// TwinCAT 3 PLC project TcUnit
// Title: TcUnit
// Company: www.tcunit.org
// Author: Jakob Sagatowski and contributors
// ProjectVersion: 1.3.2
// Description: TwinCAT unit testing framework. Documentation and examples are available at www.tcunit.org
// ProgramVersion: 3.1.4022.2
// libraries:
//   SysDir, * (System)
//   SysFile, * (System)
//   Tc2_Standard, * (Beckhoff Automation GmbH)
//   Tc2_System, * (Beckhoff Automation GmbH)
//   Tc2_Utilities, * (Beckhoff Automation GmbH)
//   Base Interfaces,newest,System
// project tree:
//   DUTs/ E_AssertionType.TcDUT, E_XmlError.TcDUT, ST_AdsLogStringMessage.TcDUT, ST_AssertResult.TcDUT, ST_AssertResultInstances.TcDUT, ST_AssertArrayResult.TcDUT, ST_AssertArrayResultInstances.TcDUT, ST_TestCaseResult.TcDUT, ST_TestSuiteResult.TcDUT, ST_TestSuiteResults.TcDUT, U_ExpectedOrActual.TcDUT
//   GVLs/ GVL_Param_TcUnit.TcGVL, GVL_TcUnit.TcGVL
//   ITFs/ I_AssertMessageFormatter.TcIO, I_TestResultLogger.TcIO, I_TestResults.TcIO
//   POUs/ FB_AdsAssertMessageFormatter.TcPOU, FB_AdsLogStringMessageFifoQueue.TcPOU, FB_AdsTestResultLogger.TcPOU, FB_FileControl.TcPOU, FB_StreamBuffer.TcPOU, FB_xUnitXmlPublisher.TcPOU, FB_TestResults.TcPOU, FB_AdjustAssertFailureMessageToMaxAllowedLength.TcPOU, FB_AssertResultStatic.TcPOU, FB_AssertArrayResultStatic.TcPOU, FB_TcUnitRunner.TcPOU, FB_Test.TcPOU, FB_TestSuite.TcPOU, FB_XmlControl.TcPOU
//   POUs/Functions/ F_AnyToUnionValue.TcPOU, F_AnyTypeClassToString.TcPOU, F_AssertionTypeToString.TcPOU, F_GetCpuCounterAs64bit.TcPOU, F_GetTestSuiteNameFromTestInstancePath.TcPOU, F_IsAnyEqualToUnionValue.TcPOU, F_RemoveInstancePathAndProjectNameFromTestInstancePath.TcPOU, IS_TEST_FINISHED.TcPOU, RUN.TcPOU, RUN_IN_SEQUENCE.TcPOU, TCUNIT_ADSLOGSTR.TcPOU, TEST.TcPOU, TEST_FINISHED.TcPOU, TEST_FINISHED_NAMED.TcPOU, TEST_ORDERED.TcPOU
//   POUs/Functions/WRITE_PROTECTED_/ WRITE_PROTECTED_BOOL.TcPOU, WRITE_PROTECTED_BYTE.TcPOU, WRITE_PROTECTED_DATE.TcPOU, WRITE_PROTECTED_DATE_AND_TIME.TcPOU, WRITE_PROTECTED_DINT.TcPOU, WRITE_PROTECTED_DWORD.TcPOU, WRITE_PROTECTED_INT.TcPOU, WRITE_PROTECTED_LREAL.TcPOU, WRITE_PROTECTED_REAL.TcPOU, WRITE_PROTECTED_SINT.TcPOU, WRITE_PROTECTED_STRING.TcPOU, WRITE_PROTECTED_WSTRING.TcPOU, WRITE_PROTECTED_TIME.TcPOU, WRITE_PROTECTED_TIME_OF_DAY.TcPOU, WRITE_PROTECTED_UDINT.TcPOU, WRITE_PROTECTED_UINT.TcPOU, WRITE_PROTECTED_ULINT.TcPOU, WRITE_PROTECTED_LWORD.TcPOU, WRITE_PROTECTED_LINT.TcPOU, WRITE_PROTECTED_USINT.TcPOU, WRITE_PROTECTED_WORD.TcPOU
//   Version/ Global_Version.TcGVL

// ---- DUTs/E_AssertionType.TcDUT
{attribute 'qualified_only'}
{attribute 'strict'}
TYPE E_AssertionType :
(
    Type_UNDEFINED := 0,
    Type_ANY,

    // Primitive types
    Type_BOOL,
    Type_BYTE,
    Type_DATE,
    Type_DATE_AND_TIME,
    Type_DINT,
    Type_DWORD,
    Type_INT,
    Type_LINT,
    Type_LREAL,
    Type_LTIME,
    Type_LWORD,
    Type_REAL,
    Type_SINT,
    Type_STRING,
    Type_TIME,
    Type_TIME_OF_DAY,
    Type_UDINT,
    Type_UINT,
    Type_ULINT,
    Type_USINT,
    Type_WORD,
    Type_WSTRING,

    // Array types
    Type_Array2D_LREAL,
    Type_Array2D_REAL,
    Type_Array3D_LREAL,
    Type_Array3D_REAL,
    Type_Array_BOOL,
    Type_Array_BYTE,
    Type_Array_DINT,
    Type_Array_DWORD,
    Type_Array_INT,
    Type_Array_LINT,
    Type_Array_LREAL,
    Type_Array_LWORD,
    Type_Array_REAL,
    Type_Array_SINT,
    Type_Array_UDINT,
    Type_Array_UINT,
    Type_Array_ULINT,
    Type_Array_USINT,
    Type_Array_WORD
) BYTE;
END_TYPE

// ---- DUTs/E_XmlError.TcDUT
{attribute 'qualified_only'}
{attribute 'strict'}
TYPE E_XmlError :
(
    Ok := 0,
    ErrorMaxBufferLen := 1,
    ErrorStringLen := 2,
    Error := 3
) BYTE;
END_TYPE

// ---- DUTs/ST_AdsLogStringMessage.TcDUT
{attribute 'pack_mode' := '1'}
TYPE ST_AdsLogStringMessage :
STRUCT
	MsgCtrlMask : DWORD;
    MsgFmtStr : T_MaxString;
    StrArg : T_MaxString;
END_STRUCT
END_TYPE

// ---- DUTs/ST_AssertResult.TcDUT
TYPE ST_AssertResult :
STRUCT
    Expected : U_ExpectedOrActual;
    Actual : U_ExpectedOrActual;
    Message : T_MaxString;
    TestInstancePath : T_MaxString;
END_STRUCT
END_TYPE

// ---- DUTs/ST_AssertResultInstances.TcDUT
TYPE ST_AssertResultInstances :
STRUCT
    AssertResult : ST_AssertResult;
    DetectionCount : UINT; // Number of instances of the "AssertResult"
    DetectionCountThisCycle : UINT; // Number of instance of the "AssertResult" in this specific PLC-cycle
END_STRUCT
END_TYPE

// ---- DUTs/ST_AssertArrayResult.TcDUT
TYPE ST_AssertArrayResult :
STRUCT
    ExpectedsSize : UDINT; // Size in bytes of the expecteds-array
    ExpectedsTypeClass : IBaseLibrary.TypeClass; // The data type of the expecteds-array
    ActualsSize : UDINT; // Size in bytes of the actuals-array
    ActualsTypeClass : IBaseLibrary.TypeClass; // The data type of the actuals-array
    Message : T_MaxString;
    TestInstancePath : T_MaxString;
END_STRUCT
END_TYPE

// ---- DUTs/ST_AssertArrayResultInstances.TcDUT
TYPE ST_AssertArrayResultInstances :
STRUCT
    AssertArrayResult : ST_AssertArrayResult;
    DetectionCount : UINT; // Number of instances of the "AssertArrayResult"
    DetectionCountThisCycle : UINT; // Number of instance of the "AssertArrayResult" in this specific PLC-cycle
END_STRUCT
END_TYPE

// ---- DUTs/ST_TestCaseResult.TcDUT
TYPE ST_TestCaseResult :
STRUCT
    TestName : T_MaxString;
    TestClassName : T_MaxString;
    TestIsFailed : BOOL;
    TestIsSkipped : BOOL;
    FailureMessage : T_MaxString;
    FailureAssertion : Tc2_System.T_MaxString;
    FailureType : E_AssertionType;
    NumberOfAsserts : UINT;
    Duration : LREAL; // in seconds
END_STRUCT
END_TYPE

// ---- DUTs/ST_TestSuiteResult.TcDUT
TYPE ST_TestSuiteResult :
STRUCT
    Name : T_MaxString; // Full class name
    Identity : UINT(0..GVL_Param_TcUnit.MaxNumberOfTestSuites); // Should be 0..GVL_Param_TcUnit.MaxNumberOfTestSuites-1 but gives unknown compiler error
    NumberOfTests : UINT(0..GVL_Param_TcUnit.MaxNumberOfTestsForEachTestSuite);
    NumberOfFailedTests : UINT(0..GVL_Param_TcUnit.MaxNumberOfTestsForEachTestSuite);
    Duration : LREAL; // In seconds
    TestCaseResults : ARRAY[1..GVL_Param_TcUnit.MaxNumberOfTestsForEachTestSuite] OF ST_TestCaseResult;
END_STRUCT
END_TYPE

// ---- DUTs/ST_TestSuiteResults.TcDUT
TYPE ST_TestSuiteResults :
STRUCT
    // General test results
    NumberOfTestSuites : UINT; // The total number of test suites
    NumberOfTestCases : UINT; // The total number of test cases (for all test suites)
    NumberOfSuccessfulTestCases : UINT; // The total number of test cases that had all ASSERTS successful
    NumberOfFailedTestCases : UINT; // The total number of test cases that had at least one ASSERT failed
    Duration : LREAL; // Duration it took for all test suites to finish, in seconds

    // Test results for each individiual test suite
    TestSuiteResults : ARRAY[1..GVL_Param_TcUnit.MaxNumberOfTestSuites] OF ST_TestSuiteResult;
END_STRUCT
END_TYPE

// ---- DUTs/U_ExpectedOrActual.TcDUT
TYPE U_ExpectedOrActual :
UNION
    boolExpectedOrActual : BOOL;
    bitExpectedOrActual : BIT;
    byteExpectedOrActual : BYTE;
    dwordExpectedOrActual : DWORD;
    lwordExpectedOrActual : LWORD;
    stringExpectedOrActual : T_MaxString;
    udintExpectedOrActual : UDINT;
    uintExpectedOrActual : UINT;
    usintExpectedOrActual : USINT;
    sintExpectedOrActual : SINT;
    intExpectedOrActual : INT;
    wordExpectedOrActual : WORD;
    dintExpectedOrActual : DINT;
    lintExpectedOrActual : LINT;
    ulintExpectedOrActual : ULINT;
    realExpectedOrActual : REAL;
    lrealExpectedOrActual : LREAL;
    wstringExpectedOrActual : WSTRING(255);
    timeExpectedOrActual : TIME;
    ltimeExpectedOrActual : LTIME;
    dateExpectedOrActual : DATE;
    dateandtimeExpectedOrActual : DATE_AND_TIME;
    timeofdayExpectedOrActual : TIME_OF_DAY;
END_UNION
END_TYPE

// ---- GVLs/GVL_Param_TcUnit.TcGVL
{attribute 'qualified_only'}
VAR_GLOBAL CONSTANT
    MaxNumberOfTestSuites : UINT := 1000;
    MaxNumberOfTestsForEachTestSuite : UINT := 100;
    MaxNumberOfAssertsForEachTestSuite : UINT := 1000;

    (* TcUnit logs complete test results. These include:
         - Number of test suites
         - Number of tests
         - Number of successful tests
         - Number of failed tests
         - Any eventual failed assertion (with the expected & actual value plus an user defined message)
       These are all printed to the ADS logger (Visual Studio error list) marked with ERROR criticality

       On top of this TcUnit also reports some statistics/extended information with HINT/INFO criticality.
       These statistics are more detailed results of the tests. This information is used when results are
       being collected by an external software (such as TcUnit-Runner) to do for example Jenkins integration.
       This extra information however takes time to print, so by setting the following parameter to FALSE
       it will speed up TcUnit finishing. *)
    LogExtendedResults : BOOL := TRUE;

    (* Enable (TRUE) or disable (FALSE) publishing of the xUnit Xml report *)
    xUnitEnablePublish : BOOL := FALSE;

    (* Default reserved PLC memory buffer used for composition of the xUnit xml file (64 kb default) *)
    xUnitBufferSize : UDINT := 65535;

    (* Default path and filename for the xunit testresults e.g.: for use with jenkins 

	   Use environment variables for a OS independent file path
	   - %TC_BOOTPRJPATH% -> 'C:\TwinCAT\3.1\Boot\' (Windows), '/usr/local/etc/TwinCAT/3.1/Boot/' (TC/BSD), '\Hard Disk\TwinCAT\3.1\Boot\' (Windows CE)
      - %TC_INSTALLPATH% -> 'C:\TwinCAT\3.1\' (Windows), '/usr/local/etc/TwinCAT/3.1/' (TC/BSD), '\Hard Disk\TwinCAT\3.1\' (Windows CE) *)
    xUnitFilePath : T_MaxString := '%TC_BOOTPRJPATH%tcunit_xunit_testresults.xml';

    (* This is the maximum number of ADS-messages that can be stored for reporting at the same time.
       Having a size of 2000 means that it's possible to report up to ~400 test cases in one single
       PLC cycle. Each entry consumes around 500 bytes, so with an example of a ring buffer size of
       2000 it means that TcUnit will consume around 1 MB of router memory. *) 
    AdsLogMessageFifoRingBufferSize : UINT := 2000;

    (* Time delay between a test suite is finished and the execution of the next test suite starts
       if using RUN_IN_SEQUENCE() *)
    TimeBetweenTestSuitesExecution : TIME := T#0MS;

    (* If TRUE, the assertion message may be printed using multiple ADS log lines. *)
    MultipleLinesPerAssertionMessage : BOOL := FALSE;
END_VAR

// ---- GVLs/GVL_TcUnit.TcGVL
{attribute 'no_assign'}
{attribute 'qualified_only'}
VAR_GLOBAL
    TcUnitRunner : FB_TcUnitRunner;

    (* Indication of whether the last instantiated test suite has an assert instance created *)
    TestSuiteIsRegistered : BOOL;

    (* Pointer to current test suite being called *)
    CurrentTestSuiteBeingCalled : POINTER TO FB_TestSuite;

    (* Current name of test being called *)
    CurrentTestNameBeingCalled : T_MaxString;

    (* Used to get the current cpu cycle counter to calculate the duration of tests and test suits, respectively *)
    GetCpuCounter : GETCPUCOUNTER;

    (* Stores the CPU cycle count with 100ns precision since the first entry into one of the Run methods (RUN, RUN_IN_SEQUENCE) *)
    StartedAt : LWORD;

    (* Duration it took for a complete run, in seconds *)
    Duration : LREAL;

    (* Whether or not the current test being called has finished running *)
    CurrentTestIsFinished : BOOL;

    (* This is a flag that indicates that the current test should be ignored, and
       thus that all assertions under it should be ignored as well. A test can be ignored either
       because the user has requested so, or because the test is a duplicate name *)
    IgnoreCurrentTest : BOOL;

    (* The assert function block instance should be 1:1 mapped to
       the test suite instance path. *)
    NumberOfInitializedTestSuites : UINT := 0;
    TestSuiteAddresses : ARRAY[1..GVL_Param_TcUnit.MaxNumberOfTestSuites] OF POINTER TO FB_TestSuite;

    (* If the user is utilizing the TEST_ORDERED(), we need to keep track of which ordered test is currently running.
       We do this by defining an array, in where we can see which current TEST_ORDERED() is the one to be handled right now.
       The below array is only used for TEST_ORDERED()-tests.  *)
    CurrentlyRunningOrderedTestInTestSuite : ARRAY[1..GVL_Param_TcUnit.MaxNumberOfTestSuites] OF UINT(1..GVL_Param_TcUnit.MaxNumberOfTestsForEachTestSuite);

    (* Buffered ADS message queue for output to the error list *)
    AdsMessageQueue : FB_AdsLogStringMessageFifoQueue;
END_VAR
VAR_GLOBAL CONSTANT
  (* Multiply a value that is given in 100ns units by this value to
     convert the value to seconds *)
  HundredNanosecondToSecond : LREAL := 1.0 / 10000000.0;
END_VAR

// ---- Version/Global_Version.TcGVL
{attribute 'TcGenerated'}
{attribute 'no-analysis'}
{attribute 'linkalways'}
// This function has been automatically generated from the project information.
VAR_GLOBAL CONSTANT
	{attribute 'const_non_replaced'}
	stLibVersion_TcUnit : ST_LibVersion := (iMajor := 1, iMinor := 3, iBuild := 2, iRevision := 0, nFlags := 0, sVersion := '1.3.2');
END_VAR

// ---- ITFs/I_AssertMessageFormatter.TcIO
INTERFACE I_AssertMessageFormatter

METHOD LogAssertFailure
VAR_INPUT
    Expected : T_MaxString;
    Actual : T_MaxString;
    Message : T_MaxString;
    TestInstancePath : T_MaxString;
END_VAR
END_METHOD

END_INTERFACE

// ---- ITFs/I_TestResultLogger.TcIO
INTERFACE I_TestResultLogger

METHOD PUBLIC LogTestSuiteResults
END_METHOD

END_INTERFACE

// ---- ITFs/I_TestResults.TcIO
INTERFACE I_TestResults

METHOD GetAreTestResultsAvailable : BOOL
END_METHOD

METHOD GetTestSuiteResults : REFERENCE TO ST_TestSuiteResults;
END_METHOD

END_INTERFACE

// ---- POUs/Functions/TEST.TcPOU
// This function declares a new test (if it has not been already declared in an earlier cycle)
FUNCTION TEST
VAR_INPUT
    TestName : T_MaxString;
END_VAR
VAR
    CounterTestSuiteAddress : UINT;
    Test : REFERENCE TO FB_Test;
END_VAR

TestName := F_LTrim(in := F_RTrim(in := TestName));

// Mark this test as the current one being executed
GVL_TcUnit.CurrentTestNameBeingCalled := TestName;

(* Check if combination of address for the test suite and test name already exists.
   For every test suite the name of the test case needs to be unique.
   If a test with this name already exists, don't add it to the available tests.
   Otherwise, add it to the available tests *)

FOR CounterTestSuiteAddress := 1 TO GVL_TcUnit.NumberOfInitializedTestSuites BY 1 DO
    // Look for the test suite by comparing to the one that is currently running
    IF GVL_TcUnit.TestSuiteAddresses[CounterTestSuiteAddress] = GVL_TcUnit.CurrentTestSuiteBeingCalled THEN
        Test REF= GVL_TcUnit.TestSuiteAddresses[CounterTestSuiteAddress]^.AddTest(TestName := TestName, IsTestOrdered := FALSE);
        GVL_TcUnit.CurrentTestIsFinished := GVL_TcUnit.TestSuiteAddresses[CounterTestSuiteAddress]^.IsTestFinished(TestName := TestName);
        IF __ISVALIDREF(Test) THEN
			Test.SetStartedAtIfNotSet(Timestamp := F_GetCpuCounterAs64bit(GVL_TcUnit.GetCpuCounter));
        END_IF
        RETURN;
    END_IF
END_FOR

END_FUNCTION

// ---- POUs/FB_Test.TcPOU
// This function block holds all data that defines a test.
FUNCTION_BLOCK FB_Test
VAR
    TestName : T_MaxString;
    TestIsFinished : BOOL;
    TestIsSkipped : BOOL; // This is set to true, if test is disabled (by putting the string "disabled_" in front of the test name
    NumberOfAssertions : UINT;

    (* In which order/sequence relative to the order tests should this test be executed/evaluated.
       A value of 0 means it is not defined by TEST_ORDERED() but by un-ordered test (TEST()).
       A value <> 0 tells in which order this test will be executed/evaluated. The lower the number, the earlier it will execute. *)
    TestOrderNumber : UINT(0..GVL_Param_TcUnit.MaxNumberOfTestsForEachTestSuite); 

    // Failure parameters. If TestIsFailed is TRUE, the other parameters will hold values as well
    TestIsFailed : BOOL; // Indication of whether this test has at least one failed assert
    AssertionMessage : T_MaxString; // Assertion message for the first assertion in this test
    AssertionFailure : Tc2_System.T_MaxString; // Assertion failure for the first assertion in this test	
    AssertionType : E_AssertionType; // Assertion type for the first assertion in this test

    StartedAt : LWORD; // Temporary variable to calculate the actual duration of the test, the value holds the cpu cycle counter when a test is started in 100ns precision
    Duration : LREAL; // Duration of the test in seconds
END_VAR

METHOD INTERNAL GetAssertionFailure : Tc2_System.T_MaxString
GetAssertionFailure := AssertionFailure;
END_METHOD

METHOD INTERNAL GetAssertionMessage : T_MaxString
GetAssertionMessage := AssertionMessage;
END_METHOD

METHOD INTERNAL GetAssertionType : E_AssertionType
GetAssertionType := AssertionType;
END_METHOD

METHOD INTERNAL GetDuration : LREAL
GetDuration := Duration;
END_METHOD

METHOD INTERNAL GetName : T_MaxString;
GetName := TestName;
END_METHOD

METHOD INTERNAL GetNumberOfAssertions : UINT
GetNumberOfAssertions := NumberOfAssertions;
END_METHOD

// Gets in which order/sequence relative to the order tests should this test be executed/evaluated.
METHOD INTERNAL GetTestOrder : UINT(0..GVL_Param_TcUnit.MaxNumberOfTestsForEachTestSuite);
GetTestOrder := TestOrderNumber;
END_METHOD

METHOD INTERNAL IsFailed : BOOL
IsFailed := TestIsFailed;
END_METHOD

METHOD INTERNAL IsFinished : BOOL
IsFinished := TestIsFinished;
END_METHOD

METHOD INTERNAL IsSkipped : BOOL
IsSkipped := TestIsSkipped;
END_METHOD

(* Sets the assertion failure. If one already exists, it's not overwritten as we keep the first assertion in the test *)
METHOD INTERNAL SetAssertionFailure
VAR_INPUT
    AssertFailure : Tc2_System.T_MaxString;
END_VAR
IF Tc2_Standard.LEN(STR := AssertionFailure) = 0 THEN
    AssertionFailure := AssertFailure;
END_IF
END_METHOD

// Sets the assertion message. If one already exists, it's not overwritten as we keep the first assertion in the test
METHOD INTERNAL SetAssertionMessage
VAR_INPUT
    AssertMessage : T_MaxString;
END_VAR
IF LEN(STR := AssertionMessage) = 0 THEN
    AssertionMessage := AssertMessage;
END_IF
END_METHOD

// Sets the assertion type. If one already exists, it's not overwritten as we keep the first assertion in the test
METHOD INTERNAL SetAssertionType
VAR_INPUT
    AssertType : E_AssertionType;
END_VAR
IF AssertionType = E_AssertionType.Type_UNDEFINED THEN
    AssertionType := AssertType;
END_IF
END_METHOD

METHOD INTERNAL SetFailed
TestIsFailed := TRUE;
END_METHOD

METHOD INTERNAL SetFinishedAndDuration : BOOL
VAR_INPUT
    FinishedAt : LWORD; // CPU cycle counter with 100ns precision
END_VAR
TestIsFinished := TRUE;
Duration := LWORD_TO_LREAL(FinishedAt - StartedAt) * GVL_TcUnit.HundredNanosecondToSecond; // Seconds
END_METHOD

METHOD INTERNAL SetName
VAR_INPUT
    Name : T_MaxString;
END_VAR
TestName := Name;
END_METHOD

METHOD INTERNAL SetNumberOfAssertions
VAR_INPUT
    NoOfAssertions : UINT;
END_VAR
NumberOfAssertions := NoOfAssertions;
END_METHOD

// Sets the test case to skipped
METHOD INTERNAL SetSkipped
TestIsSkipped := TRUE;
END_METHOD

METHOD INTERNAL SetStartedAtIfNotSet
VAR_INPUT
    Timestamp : LWORD; // CPU cycle counter with 100ns precision
END_VAR
IF StartedAt = 0 THEN
    StartedAt := Timestamp;
END_IF
END_METHOD

// Sets in which order/sequence relative to the order tests should this test be executed/evaluated.
METHOD INTERNAL SetTestOrder
VAR_INPUT
    OrderNumber : UINT(0..GVL_Param_TcUnit.MaxNumberOfTestsForEachTestSuite);
END_VAR
TestOrderNumber := OrderNumber;
END_METHOD

END_FUNCTION_BLOCK

// ---- POUs/Functions/F_GetCpuCounterAs64bit.TcPOU
(* Calls the passed GETCPUCOUNTER function block and
   converts the output of the GETCPUCOUNTER function block from 2x32bit variables to a
   single 64bit variable
*)
FUNCTION F_GetCpuCounterAs64bit : LWORD
VAR_IN_OUT CONSTANT
    CpuCounter : GETCPUCOUNTER;
END_VAR

CpuCounter();
F_GetCpuCounterAs64bit := SHL(DWORD_TO_LWORD(CpuCounter.cpuCntHiDW), 32) + DWORD_TO_LWORD(CpuCounter.cpuCntLoDW);

END_FUNCTION

// ---- POUs/Functions/RUN_IN_SEQUENCE.TcPOU
(*
    This function runs all test suites that have been initialized.
    The test suites are run in sequence (one after the other).
*)
FUNCTION RUN_IN_SEQUENCE

GVL_TcUnit.TcUnitRunner.RunTestSuiteTestsInSequence(TimeBetweenTestSuitesExecution := GVL_Param_TcUnit.TimeBetweenTestSuitesExecution);

END_FUNCTION

// ---- POUs/FB_TcUnitRunner.TcPOU
// This function block is responsible for holding track of the tests and executing them.
FUNCTION_BLOCK FB_TcUnitRunner
VAR
    // Indication of whether all test suites have reported that they are finished
    AllTestSuitesFinished : BOOL := FALSE;
    AllTestSuitesFinishedTrigger : R_TRIG;

    //Test result information
    TestResults : FB_TestResults;

    (* Prints the results to ADS so that Visual Studio can display the results.
       This test result formatter can be replaced with something else than ADS *)
    AdsTestResultLogger : FB_AdsTestResultLogger(TestResults);
    TestResultLogger : I_TestResultLogger := AdsTestResultLogger;

    (* If this flag is set, it means that some external event triggered the
       request to abort running the test suites *)
    AbortRunningTestSuites : BOOL;

    // Publishes a xUnit compatible XML file
    xUnitXmlPublisher : FB_xUnitXmlPublisher(TestResults);
    XmlTestResultPublisher : I_TestResultLogger := xUnitXmlPublisher;
END_VAR

(* This function sets a flag which makes the runner stop running the tests
   in the test suites *)
METHOD INTERNAL AbortRunningTestSuiteTests
AbortRunningTestSuites := TRUE;
END_METHOD

// This runs all the test suites in parallel
METHOD INTERNAL RunTestSuiteTests
VAR
    Counter : UINT := 0;
    BusyPrinting : BOOL;
    (* We need to hold a temporary state of the statistics 
       as we don't consider the tests to be completely finished until all test suites have executed completely.
       The reason we want to do it this way is because a test suite can run over several cycles. Only once all tests
       are finished (which might take many cycles), do we gather correct statistics *)
    NumberOfTestSuitesFinished : UINT := 0;
END_VAR
IF GVL_TcUnit.StartedAt = 0 THEN
    GVL_TcUnit.StartedAt := F_GetCpuCounterAs64bit(GVL_TcUnit.GetCpuCounter);
END_IF

// Run TcUnit test suites
IF NOT AllTestSuitesFinished THEN
    IF GVL_TcUnit.NumberOfInitializedTestSuites = 0 THEN
        AllTestSuitesFinished := TRUE;
    ELSIF GVL_TcUnit.NumberOfInitializedTestSuites > 0 THEN
        FOR Counter := 1 TO GVL_TcUnit.NumberOfInitializedTestSuites BY 1 DO
            IF GVL_TcUnit.TestSuiteAddresses[Counter]^.AreAllTestsFinished() THEN
                NumberOfTestSuitesFinished := NumberOfTestSuitesFinished + 1;
            ELSE
                GVL_TcUnit.CurrentTestSuiteBeingCalled := GVL_TcUnit.TestSuiteAddresses[Counter];
				GVL_TcUnit.CurrentTestSuiteBeingCalled^.SetStartedAtIfNotSet(Timestamp := F_GetCpuCounterAs64bit(GVL_TcUnit.GetCpuCounter));
                GVL_TcUnit.CurrentTestSuiteBeingCalled^();
				// This is not an efficient way to set the duration
				IF GVL_TcUnit.TestSuiteAddresses[Counter]^.AreAllTestsFinished() THEN
					GVL_TcUnit.CurrentTestSuiteBeingCalled^.CalculateDuration(FinishedAt := F_GetCpuCounterAs64bit(GVL_TcUnit.GetCpuCounter));
				END_IF
            END_IF
        END_FOR
        (* Check if some event triggered an abortion of running the tests, in that case abort it now.
           This can be accomplished by setting the result of the test suites run to finished. *)
        IF AbortRunningTestSuites THEN
            NumberOfTestSuitesFinished := GVL_TcUnit.NumberOfInitializedTestSuites;
        END_IF

        IF NumberOfTestSuitesFinished = GVL_TcUnit.NumberOfInitializedTestSuites THEN
            AllTestSuitesFinished := TRUE;
        END_IF
    END_IF
END_IF

// Store test suite results continuously
TestResults();

// Log test suite results continuously
TestResultLogger.LogTestSuiteResults();

// Publish the xUnit Xml file once if enabled
XmlTestResultPublisher.LogTestSuiteResults();

// Run the buffered ADS logger
GVL_TcUnit.AdsMessageQueue();
END_METHOD

// This runs all the test suites in sequence (one after the other)
METHOD INTERNAL RunTestSuiteTestsInSequence
VAR_INPUT
    TimeBetweenTestSuitesExecution : TIME; // Time delay between a test suite is finished and the next test suite starts
END_VAR
VAR
    BusyPrinting : BOOL;
    (* We need to hold a temporary state of the statistics
       as we don't consider the tests to be completely finished until all test suites have executed completely.
       The reason we want to do it this way is because a test suite can run over several cycles. Only once all tests
       are finished (which might take many cycles), do we gather correct statistics *)
    NumberOfTestSuitesFinished : UINT := 0;
END_VAR
VAR_INST
    (* This variable holds which current test suite is being called, as we are running
       each one in a sequence (one by one) *)
     CurrentlyRunningTestSuite : UINT := 1;
     TimerBetweenExecutionOfTestSuites : TOF;
END_VAR
IF GVL_TcUnit.StartedAt = 0 THEN
    GVL_TcUnit.StartedAt := F_GetCpuCounterAs64bit(GVL_TcUnit.GetCpuCounter);
END_IF

TimerBetweenExecutionOfTestSuites(PT := TimeBetweenTestSuitesExecution);
// Run TcUnit test suites
IF NOT AllTestSuitesFinished THEN
    IF GVL_TcUnit.NumberOfInitializedTestSuites = 0 THEN
        AllTestSuitesFinished := TRUE;
    ELSIF GVL_TcUnit.NumberOfInitializedTestSuites > 0 THEN
        IF TimerBetweenExecutionOfTestSuites.Q THEN
            TimerBetweenExecutionOfTestSuites.IN := FALSE;
        END_IF
        IF GVL_TcUnit.TestSuiteAddresses[CurrentlyRunningTestSuite]^.AreAllTestsFinished() THEN
            IF CurrentlyRunningTestSuite <> GVL_TcUnit.NumberOfInitializedTestSuites THEN
                NumberOfTestSuitesFinished := NumberOfTestSuitesFinished + 1;
                CurrentlyRunningTestSuite := CurrentlyRunningTestSuite + 1;
                TimerBetweenExecutionOfTestSuites.IN := TRUE;
				GVL_TcUnit.CurrentTestSuiteBeingCalled^.CalculateDuration(FinishedAt := F_GetCpuCounterAs64bit(GVL_TcUnit.GetCpuCounter));
            END_IF
        ELSIF NOT TimerBetweenExecutionOfTestSuites.Q THEN
            GVL_TcUnit.CurrentTestSuiteBeingCalled := GVL_TcUnit.TestSuiteAddresses[CurrentlyRunningTestSuite];
			GVL_TcUnit.CurrentTestSuiteBeingCalled^.SetStartedAtIfNotSet(Timestamp := F_GetCpuCounterAs64bit(GVL_TcUnit.GetCpuCounter));
            GVL_TcUnit.CurrentTestSuiteBeingCalled^();
			// This is not an efficient way to set the duration
			IF GVL_TcUnit.TestSuiteAddresses[CurrentlyRunningTestSuite]^.AreAllTestsFinished() THEN
				GVL_TcUnit.CurrentTestSuiteBeingCalled^.CalculateDuration(FinishedAt := F_GetCpuCounterAs64bit(GVL_TcUnit.GetCpuCounter));
			END_IF
        END_IF
        (* Check if some event triggered an abortion of running the tests, in that case abort it now.
           This can be accomplished by setting the result of the test suites run to finished. *)
        IF AbortRunningTestSuites THEN
            NumberOfTestSuitesFinished := GVL_TcUnit.NumberOfInitializedTestSuites;
        END_IF
        IF NumberOfTestSuitesFinished = GVL_TcUnit.NumberOfInitializedTestSuites THEN
            AllTestSuitesFinished := TRUE;
        END_IF
    END_IF
END_IF

// Store test suite results continuously
TestResults();

// Log test suite results continuously
TestResultLogger.LogTestSuiteResults();

// Publish the xUnit Xml file once if enabled
XmlTestResultPublisher.LogTestSuiteResults();

// Run the buffered ADS logger
GVL_TcUnit.AdsMessageQueue();
END_METHOD

END_FUNCTION_BLOCK

// ---- POUs/FB_TestResults.TcPOU
// This function block holds results of the complete test run, i.e. results for all test suites
FUNCTION_BLOCK FB_TestResults IMPLEMENTS I_TestResults
VAR
    // Test results
    TestSuiteResults : ST_TestSuiteResults;

    // Misc variables
    StoringTestSuiteResultNumber : UINT(1..GVL_Param_TcUnit.MaxNumberOfTestSuites);
    StoringTestSuiteTrigger : R_TRIG;
    StoredTestSuiteResults : BOOL;
    StoredGeneralTestResults : BOOL;
    NumberOfTestsToAnalyse : UINT(1..GVL_Param_TcUnit.MaxNumberOfTestsForEachTestSuite);
END_VAR
VAR_TEMP
    TestSuiteName : T_MaxString;
    TestName : T_MaxString;

    TestsInTestSuiteCounter : UINT(1..GVL_Param_TcUnit.MaxNumberOfTestsForEachTestSuite);

    TestToBeStored : FB_Test;
    GeneralTestResultsTestSuitesCounter : UINT(1..GVL_Param_TcUnit.MaxNumberOfTestSuites);
END_VAR

// The body of the function block stores the test results
IF StoringTestSuiteResultNumber <= GVL_TcUnit.NumberOfInitializedTestSuites AND NOT StoredTestSuiteResults THEN
	StoringTestSuiteTrigger(CLK := GVL_TcUnit.TestSuiteAddresses[StoringTestSuiteResultNumber]^.AreAllTestsFinished());

    IF StoringTestSuiteTrigger.Q THEN
        // Remove everything except the program name + "." + test suite name
        TestSuiteName := F_RemoveInstancePathAndProjectNameFromTestInstancePath(TestInstancePath := GVL_TcUnit.TestSuiteAddresses[StoringTestSuiteResultNumber]^.GetInstancePath());

        // Store test suite name and ID
        TestSuiteResults.TestSuiteResults[StoringTestSuiteResultNumber].Name := TestSuiteName;
        TestSuiteResults.TestSuiteResults[StoringTestSuiteResultNumber].Identity := StoringTestSuiteResultNumber - 1;

        // Store number of tests in test suite
        TestSuiteResults.TestSuiteResults[StoringTestSuiteResultNumber].NumberOfTests :=
            GVL_TcUnit.TestSuiteAddresses[StoringTestSuiteResultNumber]^.GetNumberOfTests();

        // Store number of failed tests in test suite
        TestSuiteResults.TestSuiteResults[StoringTestSuiteResultNumber].NumberOfFailedTests :=
            GVL_TcUnit.TestSuiteAddresses[StoringTestSuiteResultNumber]^.GetNumberOfFailedTests();

        // Store the duration
        TestSuiteResults.TestSuiteResults[StoringTestSuiteResultNumber].Duration :=
            GVL_TcUnit.TestSuiteAddresses[StoringTestSuiteResultNumber]^.GetDuration();

        // Limit the test analyse to the max array limit of 'Tests[]' in FB_TestSuite
        NumberOfTestsToAnalyse := GVL_TcUnit.TestSuiteAddresses[StoringTestSuiteResultNumber]^.GetNumberOfTestsToAnalyse();

        // Iterate and print all tests in test suite
        FOR TestsInTestSuiteCounter := 1 TO NumberOfTestsToAnalyse BY 1 DO
            TestToBeStored := GVL_TcUnit.TestSuiteAddresses[StoringTestSuiteResultNumber]^.GetTestByPosition(TestsInTestSuiteCounter);
            // Store test name
            TestSuiteResults.TestSuiteResults[StoringTestSuiteResultNumber].TestCaseResults[TestsInTestSuiteCounter].TestName := TestToBeStored.GetName();

            // Store test class name
            TestSuiteResults.TestSuiteResults[StoringTestSuiteResultNumber].TestCaseResults[TestsInTestSuiteCounter].TestClassName :=
                F_RemoveInstancePathAndProjectNameFromTestInstancePath(GVL_TcUnit.TestSuiteAddresses[StoringTestSuiteResultNumber]^.GetInstancePath());

            // Store whether the test has failed
            TestSuiteResults.TestSuiteResults[StoringTestSuiteResultNumber].TestCaseResults[TestsInTestSuiteCounter].TestIsFailed :=
                TestToBeStored.IsFailed();

            // Store whether the test was skipped
            TestSuiteResults.TestSuiteResults[StoringTestSuiteResultNumber].TestCaseResults[TestsInTestSuiteCounter].TestIsSkipped :=
                TestToBeStored.IsSkipped();

            // Store the (first failed) assertion message
            TestSuiteResults.TestSuiteResults[StoringTestSuiteResultNumber].TestCaseResults[TestsInTestSuiteCounter].FailureMessage :=
                TestToBeStored.GetAssertionMessage();
                
            (* Store the (first failed) assertion failure *)
            TestSuiteResults.TestSuiteResults[StoringTestSuiteResultNumber].TestCaseResults[TestsInTestSuiteCounter].FailureAssertion :=
                TestToBeStored.GetAssertionFailure();

            // Store the (first failed) assertion type
            TestSuiteResults.TestSuiteResults[StoringTestSuiteResultNumber].TestCaseResults[TestsInTestSuiteCounter].FailureType :=
                TestToBeStored.GetAssertionType();

            // Store number of assertions made
            TestSuiteResults.TestSuiteResults[StoringTestSuiteResultNumber].TestCaseResults[TestsInTestSuiteCounter].NumberOfAsserts :=
                TestToBeStored.GetNumberOfAssertions();

            // Store the duration of the test
            TestSuiteResults.TestSuiteResults[StoringTestSuiteResultNumber].TestCaseResults[TestsInTestSuiteCounter].Duration :=
                TestToBeStored.GetDuration();
        END_FOR

        IF StoringTestSuiteResultNumber = GVL_TcUnit.NumberOfInitializedTestSuites THEN
            StoredTestSuiteResults := TRUE;
        ELSE
            StoringTestSuiteResultNumber := StoringTestSuiteResultNumber + 1;
        END_IF
        StoringTestSuiteTrigger(CLK := FALSE); // Reset trigger
    END_IF
END_IF

(* If all test suites have finished running, store the general test results.
   Take care OF the special CASE where no tests have NOT yet been defined *)
IF GVL_TcUnit.NumberOfInitializedTestSuites = 0 AND (NOT StoredGeneralTestResults) THEN
    StoredGeneralTestResults := TRUE;
    StoredTestSuiteResults := TRUE;
ELSIF StoringTestSuiteResultNumber = GVL_TcUnit.NumberOfInitializedTestSuites AND_THEN
    GVL_TcUnit.TestSuiteAddresses[StoringTestSuiteResultNumber]^.AreAllTestsFinished() AND StoredTestSuiteResults AND (NOT StoredGeneralTestResults) THEN
    TestSuiteResults.NumberOfTestSuites := GVL_TcUnit.NumberOfInitializedTestSuites;
	GVL_TcUnit.Duration := LWORD_TO_LREAL(F_GetCpuCounterAs64bit(GVL_TcUnit.GetCpuCounter) - GVL_TcUnit.StartedAt) * GVL_TcUnit.HundredNanosecondToSecond; // Seconds
    TestSuiteResults.Duration := GVL_TcUnit.Duration;
    FOR GeneralTestResultsTestSuitesCounter := 1 TO GVL_TcUnit.NumberOfInitializedTestSuites BY 1 DO
        TestSuiteResults.NumberOfTestCases := TestSuiteResults.NumberOfTestCases + TestSuiteResults.TestSuiteResults[GeneralTestResultsTestSuitesCounter].NumberOfTests;
        TestSuiteResults.NumberOfSuccessfulTestCases := TestSuiteResults.NumberOfSuccessfulTestCases +
                                                        (TestSuiteResults.TestSuiteResults[GeneralTestResultsTestSuitesCounter].NumberOfTests -
                                                         TestSuiteResults.TestSuiteResults[GeneralTestResultsTestSuitesCounter].NumberOfFailedTests);
        TestSuiteResults.NumberOfFailedTestCases := TestSuiteResults.NumberOfFailedTestCases + TestSuiteResults.TestSuiteResults[GeneralTestResultsTestSuitesCounter].NumberOfFailedTests;
    END_FOR
    StoredGeneralTestResults := TRUE;
END_IF

// Returns whether the storing of the test results is finished
METHOD PUBLIC GetAreTestResultsAvailable : BOOL
GetAreTestResultsAvailable := (StoredTestSuiteResults AND StoredGeneralTestResults);
END_METHOD

METHOD PUBLIC GetTestSuiteResults : REFERENCE TO ST_TestSuiteResults;
GetTestSuiteResults REF=TestSuiteResults;
END_METHOD

END_FUNCTION_BLOCK

// ---- POUs/Functions/F_RemoveInstancePathAndProjectNameFromTestInstancePath.TcPOU
FUNCTION F_RemoveInstancePathAndProjectNameFromTestInstancePath : T_MaxString
VAR_INPUT
    TestInstancePath : T_MaxString;
END_VAR
VAR
    CharacterPositionOfProjectName : INT;
    ProjectNameWithDot : T_MaxString;
END_VAR

// Add the '.' character to the project name for search
ProjectNameWithDot := CONCAT(STR1 := TwinCAT_SystemInfoVarList._AppInfo.ProjectName, STR2 := '.');

// Find the character position of the beginning of the first occurence of the project name
CharacterPositionOfProjectName := FIND(STR1 := TestInstancePath, STR2 := ProjectNameWithDot);

IF CharacterPositionOfProjectName > 0 THEN
    TestInstancePath := DELETE(STR := TestInstancePath,
                               LEN := CharacterPositionOfProjectName-1 + LEN(ProjectNameWithDot),
                               POS := 1);
END_IF

// Check if the project name happens to be the same as namespace, and in that case, remove that as well
CharacterPositionOfProjectName := FIND(STR1 := TestInstancePath,
                                                    STR2 := ProjectNameWithDot);

IF CharacterPositionOfProjectName > 0 THEN
    TestInstancePath := DELETE(STR := TestInstancePath,
                               LEN := CharacterPositionOfProjectName - 1 +  LEN(STR := ProjectNameWithDot),
                               POS := 1);
END_IF

F_RemoveInstancePathAndProjectNameFromTestInstancePath := TestInstancePath;

END_FUNCTION

// ---- POUs/FB_AdsTestResultLogger.TcPOU
(*
    This function block reports the results from the tests using the built-in ADSLOGSTR functionality
    provided by the Tc2_System library. This sends the result using ADS, which is consumed by the "Error List"
    of Visual Studio (which can print Errors, Warnings and Messages).
*)
FUNCTION_BLOCK FB_AdsTestResultLogger IMPLEMENTS I_TestResultLogger
VAR
    TestResults : I_TestResults;

    PrintingTestSuiteResultNumber : UINT(1..GVL_Param_TcUnit.MaxNumberOfTestSuites);
    PrintingTestSuiteTrigger : R_TRIG;

    // This flag is set once the final end result has printed
    PrintedFinalTestResults : BOOL;

    // This flag is set once the test suites result have been printed
    PrintedTestSuitesResults : BOOL;
END_VAR

METHOD FB_init : BOOL
VAR_INPUT
	bInitRetains : BOOL; // if TRUE, the retain variables are initialized (warm start / cold start)
	bInCopyCode : BOOL;  // if TRUE, the instance afterwards gets moved into the copy code (online change)
    iTestResults : I_TestResults;
END_VAR
TestResults := iTestResults;
END_METHOD

METHOD PUBLIC LogTestSuiteResults
VAR
    TcUnitTestResults : REFERENCE TO ST_TestSuiteResults;
    StringToPrint : T_MaxString; 
    TestsInTestSuiteCounter : UINT(1..GVL_Param_TcUnit.MaxNumberOfTestsForEachTestSuite);
    MaxNumberOfTestsToPrint : UINT(1..GVL_Param_TcUnit.MaxNumberOfTestsForEachTestSuite);
END_VAR
VAR CONSTANT
    TEST_STATUS_SKIP : STRING := 'SKIP';
    TEST_STATUS_PASS : STRING := 'PASS';
    TEST_STATUS_FAIL : STRING := 'FAIL';
END_VAR
TcUnitTestResults REF= TestResults.GetTestSuiteResults();

IF PrintingTestSuiteResultNumber <= GVL_TcUnit.NumberOfInitializedTestSuites AND_THEN NOT PrintedTestSuitesResults THEN
    PrintingTestSuiteTrigger(CLK := GVL_TcUnit.TestSuiteAddresses[PrintingTestSuiteResultNumber]^.AreAllTestsFinished());
    IF PrintingTestSuiteTrigger.Q THEN
        StringToPrint := CONCAT(STR1 := '| Test suite ID=',
                                STR2 := UINT_TO_STRING(TcUnitTestResults.TestSuiteResults[PrintingTestSuiteResultNumber].Identity));
        StringToPrint := CONCAT(STR1 := StringToPrint,
                                STR2 :=  ' $'%s$'');

        // Print test suite name and ID
        GVL_TcUnit.AdsMessageQueue.WriteLog(MsgCtrlMask := ADSLOG_MSGTYPE_HINT,
                                            MsgFmtStr := StringToPrint,
                                            StrArg := TcUnitTestResults.TestSuiteResults[PrintingTestSuiteResultNumber].Name);

        // Print number of tests/number of failed tests in test suite
        StringToPrint := CONCAT(STR1 := '| ID=',
                                             STR2 := UINT_TO_STRING(TcUnitTestResults.TestSuiteResults[PrintingTestSuiteResultNumber].Identity));
        StringToPrint := CONCAT(STR1 := StringToPrint,
                                             STR2 := ' number of tests=');
        StringToPrint := CONCAT(STR1 := StringToPrint,
                                             STR2 := UINT_TO_STRING(TcUnitTestResults.TestSuiteResults[PrintingTestSuiteResultNumber].NumberOfTests));
        StringToPrint := CONCAT(STR1 := StringToPrint,
                                             STR2 := ', number of failed tests=');
        StringToPrint := CONCAT(STR1 := StringToPrint,
                                             STR2 := UINT_TO_STRING(TcUnitTestResults.TestSuiteResults[PrintingTestSuiteResultNumber].NumberOfFailedTests));
        StringToPrint := CONCAT(STR1 := StringToPrint,
                                             STR2 := ', duration=');
        StringToPrint := CONCAT(STR1 := StringToPrint,
                                             STR2 := LREAL_TO_STRING(TcUnitTestResults.TestSuiteResults[PrintingTestSuiteResultNumber].Duration));
											 
        GVL_TcUnit.AdsMessageQueue.WriteLog(MsgCtrlMask := ADSLOG_MSGTYPE_HINT,
                                            MsgFmtStr := StringToPrint,
                                            StrArg := '');

        // Print error if there are too many tests in the test suite
        IF (TcUnitTestResults.TestSuiteResults[PrintingTestSuiteResultNumber].NumberOfTests > GVL_Param_TcUnit.MaxNumberOfTestsForEachTestSuite) THEN
            MaxNumberOfTestsToPrint := GVL_Param_TcUnit.MaxNumberOfTestsForEachTestSuite;
        ELSE
            MaxNumberOfTestsToPrint := TcUnitTestResults.TestSuiteResults[PrintingTestSuiteResultNumber].NumberOfTests;
        END_IF

        // Iterate and print all tests in test suite
        FOR TestsInTestSuiteCounter := 1 TO MaxNumberOfTestsToPrint BY 1 DO
            // Print test name
            GVL_TcUnit.AdsMessageQueue.WriteLog(MsgCtrlMask := ADSLOG_MSGTYPE_HINT,
                                                MsgFmtStr := '| Test name=%s',
                                                StrArg := TcUnitTestResults.TestSuiteResults[PrintingTestSuiteResultNumber].TestCaseResults[TestsInTestSuiteCounter].TestName);
            // Print test class name
            GVL_TcUnit.AdsMessageQueue.WriteLog(MsgCtrlMask := ADSLOG_MSGTYPE_HINT,
                                                MsgFmtStr := '| Test class name=%s',
                                                StrArg := TcUnitTestResults.TestSuiteResults[PrintingTestSuiteResultNumber].TestCaseResults[TestsInTestSuiteCounter].TestClassName);

            // Print test result/status (SUCCESS, FAILED, SKIPPED) + number of assertions made
            IF TcUnitTestResults.TestSuiteResults[PrintingTestSuiteResultNumber].TestCaseResults[TestsInTestSuiteCounter].TestIsFailed THEN
                StringToPrint := CONCAT(STR1 := '| Test status=', STR2 := TEST_STATUS_FAIL);
            ELSIF TcUnitTestResults.TestSuiteResults[PrintingTestSuiteResultNumber].TestCaseResults[TestsInTestSuiteCounter].TestIsSkipped THEN
                StringToPrint := CONCAT(STR1 := '| Test status=', STR2 := TEST_STATUS_SKIP);
            ELSE
                StringToPrint := CONCAT(STR1 := '| Test status=', STR2 := TEST_STATUS_PASS);
            END_IF

            StringToPrint := CONCAT(STR1 := StringToPrint, STR2 := ', number of asserts=');
            StringToPrint := CONCAT(STR1 := StringToPrint, STR2 :=
                                                 UINT_TO_STRING(TcUnitTestResults.TestSuiteResults[PrintingTestSuiteResultNumber].TestCaseResults[TestsInTestSuiteCounter].NumberOfAsserts));
            StringToPrint := CONCAT(STR1 := StringToPrint, STR2 := ', duration=');
            StringToPrint := CONCAT(STR1 := StringToPrint, STR2 :=
                                                 LREAL_TO_STRING(TcUnitTestResults.TestSuiteResults[PrintingTestSuiteResultNumber].TestCaseResults[TestsInTestSuiteCounter].Duration));												 
            GVL_TcUnit.AdsMessageQueue.WriteLog(MsgCtrlMask := ADSLOG_MSGTYPE_HINT,
                                                MsgFmtStr := StringToPrint,
                                                StrArg := '');

            // Print assertion/failure message (if existing)
            IF (LEN(STR := TcUnitTestResults.TestSuiteResults[PrintingTestSuiteResultNumber].TestCaseResults[TestsInTestSuiteCounter].FailureMessage) > 0) THEN
                GVL_TcUnit.AdsMessageQueue.WriteLog(MsgCtrlMask := ADSLOG_MSGTYPE_HINT,
                                                    MsgFmtStr := '| Test assert message=%s',
                                                    StrArg := TcUnitTestResults.TestSuiteResults[PrintingTestSuiteResultNumber].TestCaseResults[TestsInTestSuiteCounter].FailureMessage);
            END_IF

            // Print assertion/failure type (if existing)
            IF TcUnitTestResults.TestSuiteResults[PrintingTestSuiteResultNumber].TestCaseResults[TestsInTestSuiteCounter].FailureType <> E_AssertionType.Type_UNDEFINED THEN
                GVL_TcUnit.AdsMessageQueue.WriteLog(MsgCtrlMask := ADSLOG_MSGTYPE_HINT,
                                                    MsgFmtStr := '| Test assert type=%s',
                                                    StrArg := F_AssertionTypeToString(AssertionType :=
                                                        TcUnitTestResults.TestSuiteResults[PrintingTestSuiteResultNumber].TestCaseResults[TestsInTestSuiteCounter].FailureType));
            END_IF
        END_FOR

        // Print error message if there are too many tests in the test suite
        IF (TcUnitTestResults.TestSuiteResults[PrintingTestSuiteResultNumber].NumberOfTests > GVL_Param_TcUnit.MaxNumberOfTestsForEachTestSuite) THEN
            GVL_TcUnit.AdsMessageQueue.WriteLog(MsgCtrlMask := ADSLOG_MSGTYPE_ERROR,
                                                MsgFmtStr := 'Tests failed because the number of tests (%s',
                                                StrArg := CONCAT(STR1 := TO_STRING(TcUnitTestResults.TestSuiteResults[PrintingTestSuiteResultNumber].NumberOfTests),
                                                                              STR2 := CONCAT(STR1 := ') in the test suite $'',
                                                                                                          STR2 := CONCAT(STR1 := TcUnitTestResults.TestSuiteResults[PrintingTestSuiteResultNumber].Name,
                                                                                                                                      STR2 := CONCAT(STR1 := '$' are more than is defined in parameter $'GVL_Param_TcUnit.MaxNumberOfTestsForEachTestSuite$' (',
                                                                                                                                                                  STR2 := CONCAT(STR1 := UINT_TO_STRING(GVL_Param_TcUnit.MaxNumberOfTestsForEachTestSuite),
                                                                                                                                                                                              STR2 := '). Please increase this parameter.'))))));
        END_IF

        IF PrintingTestSuiteResultNumber = GVL_TcUnit.NumberOfInitializedTestSuites THEN
            PrintedTestSuitesResults := TRUE;
        ELSE
            PrintingTestSuiteResultNumber := PrintingTestSuiteResultNumber + 1;
        END_IF
        PrintingTestSuiteTrigger(CLK := FALSE); // Reset trigger
    END_IF
END_IF

// Log end results once all test suites have finished running
IF (GVL_TcUnit.NumberOfInitializedTestSuites = 0 OR PrintingTestSuiteResultNumber = GVL_TcUnit.NumberOfInitializedTestSuites)
    AND NOT PrintedFinalTestResults AND TestResults.GetAreTestResultsAvailable() THEN
    GVL_TcUnit.AdsMessageQueue.WriteLog(MsgCtrlMask := ADSLOG_MSGTYPE_ERROR,
                                        MsgFmtStr := '%s',
                                        StrArg := '| ==========TESTS FINISHED RUNNING==========');
    GVL_TcUnit.AdsMessageQueue.WriteLog(MsgCtrlMask := ADSLOG_MSGTYPE_ERROR,
                                        MsgFmtStr := '| Test suites: %s',
                                        StrArg := UINT_TO_STRING(TcUnitTestResults.NumberOfTestSuites));
    GVL_TcUnit.AdsMessageQueue.WriteLog(MsgCtrlMask := ADSLOG_MSGTYPE_ERROR,
                                        MsgFmtStr := '| Tests: %s',
                                        StrArg := UINT_TO_STRING(TcUnitTestResults.NumberOfTestCases));
    GVL_TcUnit.AdsMessageQueue.WriteLog(MsgCtrlMask := ADSLOG_MSGTYPE_ERROR,
                                        MsgFmtStr := '| Successful tests: %s',
                                        StrArg := UINT_TO_STRING(TcUnitTestResults.NumberOfSuccessfulTestCases));
    GVL_TcUnit.AdsMessageQueue.WriteLog(MsgCtrlMask := ADSLOG_MSGTYPE_ERROR,
                                        MsgFmtStr := '| Failed tests: %s',
                                        StrArg := UINT_TO_STRING(TcUnitTestResults.NumberOfFailedTestCases));
    GVL_TcUnit.AdsMessageQueue.WriteLog(MsgCtrlMask := ADSLOG_MSGTYPE_ERROR,
                                        MsgFmtStr := '| Duration: %s',
                                        StrArg := LREAL_TO_STRING(TcUnitTestResults.Duration));                                        
    GVL_TcUnit.AdsMessageQueue.WriteLog(MsgCtrlMask := ADSLOG_MSGTYPE_ERROR,
                                        MsgFmtStr := '%s',
                                        StrArg := '| ======================================');
    PrintedFinalTestResults := TRUE;
END_IF
END_METHOD

END_FUNCTION_BLOCK

// ---- POUs/Functions/F_AssertionTypeToString.TcPOU
(* Since TwinCAT 3.1.4024.x it's possible to do TO_STRING on enumerations,
   but for backward compability we need to do it manually *)
FUNCTION F_AssertionTypeToString : T_MaxString
VAR_INPUT
    AssertionType : E_AssertionType;
END_VAR

CASE AssertionType OF
    E_AssertionType.Type_UNDEFINED :
        F_AssertionTypeToString := 'UNDEFINED';

    E_AssertionType.Type_ANY :
        F_AssertionTypeToString := 'ANY';

    (* Primitive types *)
    E_AssertionType.Type_BOOL :
        F_AssertionTypeToString := 'BOOL';

    E_AssertionType.Type_BYTE :
        F_AssertionTypeToString := 'BYTE';

    E_AssertionType.Type_DATE :
        F_AssertionTypeToString := 'DATE';

    E_AssertionType.Type_DATE_AND_TIME :
        F_AssertionTypeToString := 'DATE_AND_TIME';

    E_AssertionType.Type_DINT :
        F_AssertionTypeToString := 'DINT';

    E_AssertionType.Type_DWORD :
        F_AssertionTypeToString := 'DWORD';

    E_AssertionType.Type_INT :
        F_AssertionTypeToString := 'INT';

    E_AssertionType.Type_LINT :
        F_AssertionTypeToString := 'LINT';

    E_AssertionType.Type_LREAL :
        F_AssertionTypeToString := 'LREAL';

    E_AssertionType.Type_LTIME :
        F_AssertionTypeToString := 'LTIME';

    E_AssertionType.Type_LWORD :
        F_AssertionTypeToString := 'LWORD';

    E_AssertionType.Type_REAL :
        F_AssertionTypeToString := 'REAL';

    E_AssertionType.Type_SINT :
        F_AssertionTypeToString := 'SINT';

    E_AssertionType.Type_STRING :
        F_AssertionTypeToString := 'STRING';

    E_AssertionType.Type_TIME :
        F_AssertionTypeToString := 'TIME';

    E_AssertionType.Type_TIME_OF_DAY :
        F_AssertionTypeToString := 'TIME_OF_DAY';

    E_AssertionType.Type_UDINT :
        F_AssertionTypeToString := 'UDINT';

    E_AssertionType.Type_UINT :
        F_AssertionTypeToString := 'UINT';

    E_AssertionType.Type_ULINT :
        F_AssertionTypeToString := 'ULINT';

    E_AssertionType.Type_USINT :
        F_AssertionTypeToString := 'USINT';

    E_AssertionType.Type_WORD :
        F_AssertionTypeToString := 'WORD';

    E_AssertionType.Type_WSTRING :
        F_AssertionTypeToString := 'WSTRING';


    (* Array types *)
    E_AssertionType.Type_Array2D_LREAL :
        F_AssertionTypeToString := 'Array2D_LREAL';

    E_AssertionType.Type_Array2D_REAL :
        F_AssertionTypeToString := 'Array2D_REAL';

    E_AssertionType.Type_Array3D_LREAL :
        F_AssertionTypeToString := 'Array3D_LREAL';

    E_AssertionType.Type_Array3D_REAL :
        F_AssertionTypeToString := 'Array3D_REAL';

    E_AssertionType.Type_Array_BOOL :
        F_AssertionTypeToString := 'Array_BOOL';

    E_AssertionType.Type_Array_BYTE :
        F_AssertionTypeToString := 'Array_BYTE';

    E_AssertionType.Type_Array_DINT :
        F_AssertionTypeToString := 'Array_DINT';

    E_AssertionType.Type_Array_DWORD :
        F_AssertionTypeToString := 'Array_DWORD';

    E_AssertionType.Type_Array_INT :
        F_AssertionTypeToString := 'Array_INT';

    E_AssertionType.Type_Array_LINT :
        F_AssertionTypeToString := 'Array_LINT';

    E_AssertionType.Type_Array_LREAL :
        F_AssertionTypeToString := 'Array_LREAL';

    E_AssertionType.Type_Array_LWORD :
        F_AssertionTypeToString := 'Array_LWORD';

    E_AssertionType.Type_Array_REAL :
        F_AssertionTypeToString := 'Array_REAL';

    E_AssertionType.Type_Array_SINT :
        F_AssertionTypeToString := 'Array_SINT';

    E_AssertionType.Type_Array_UDINT :
        F_AssertionTypeToString := 'Array_UDINT';

    E_AssertionType.Type_Array_UINT :
        F_AssertionTypeToString := 'Array_UINT';

    E_AssertionType.Type_Array_ULINT :
        F_AssertionTypeToString := 'Array_ULINT';

    E_AssertionType.Type_Array_USINT :
        F_AssertionTypeToString := 'Array_USINT';

    E_AssertionType.Type_Array_WORD :
        F_AssertionTypeToString := 'Array_WORD';

    ELSE
        F_AssertionTypeToString := 'UNDEFINED';

END_CASE

END_FUNCTION

// ---- POUs/FB_xUnitXmlPublisher.TcPOU
// Publishes test results into an xUnit compatible Xml file
FUNCTION_BLOCK FB_xUnitXmlPublisher IMPLEMENTS I_TestResultLogger
VAR
    // Dependency injection via FB_Init
    _testResults : I_TestResults;

    _xmlFileStream : FB_XmlFileStream;
    _xml : FB_XMLControl(_xmlFileStream);

    _writingTestSuiteResultNumber : UINT(1..GVL_Param_TcUnit.MaxNumberOfTestSuites);
    _publishTrigger : R_TRIG;
END_VAR

(*
    FB_Init is always available implicitly AND it is used primarily FOR initialization.
    The return value is not evaluated. For a specific influence, you can also declare the
    methods explicitly and provide additional code there with the standard initialization
    code. You can evaluate the return value.
*)
METHOD FB_Init: BOOL
VAR_INPUT
    bInitRetains: BOOL; // TRUE: the retain variables are initialized (reset warm / reset cold)
    bInCopyCode: BOOL;  // TRUE: the instance will be copied to the copy code afterward (online change)
    iTestResults : I_TestResults; // Interface dependency injection
END_VAR
// Set testresult interface
THIS^._testResults := iTestResults;
END_METHOD

(*
    This method is responsible for the entire generation of the output file. 
    The output of the xml writer is NOT beautified.

    When new data is available, feel free to add it to the report
*)
METHOD PUBLIC LogTestSuiteResults
VAR
    UnitTestResults : REFERENCE TO ST_TestSuiteResults;
    CurrentSuiteNumber : UINT;
    CurrentTestCount : UINT;
END_VAR
VAR CONSTANT
    TEST_STATUS_SKIP : STRING := 'SKIP';
    TEST_STATUS_PASS : STRING := 'PASS';
    TEST_STATUS_FAIL : STRING := 'FAIL';
END_VAR
UnitTestResults REF= _testResults.GetTestSuiteResults();

// Only publish once if "GVL_Param_TcUnit.xUnitEnablePublish" is enabled and all test results are stored.
_publishTrigger(CLK := (_testResults.GetAreTestResultsAvailable() AND GVL_Param_TcUnit.xUnitEnablePublish));
IF _publishTrigger.Q THEN

    _xmlFileStream.CreateFile();  

    // <?xml version="1.0" encoding="UTF-8"?>
    _xml.WriteDocumentHeader(Header := '<?xml version="1.0" encoding="UTF-8"?>');

    // <testsuites>
    _xml.NewTag('testsuites');
    _xml.NewParameter('disabled', '');
    _xml.NewParameter('failures', UINT_TO_STRING(UnitTestResults.NumberOfFailedTestCases));
    _xml.NewParameter('tests', UINT_TO_STRING(UnitTestResults.NumberOfSuccessfulTestCases));
    _xml.NewParameter('time', LREAL_TO_STRING(UnitTestResults.Duration));

    FOR CurrentSuiteNumber := 1 TO UnitTestResults.NumberOfTestSuites BY 1 DO
        // <testsuite>
        _xml.NewTag('testsuite');
        _xml.NewParameter('id', UINT_TO_STRING(UnitTestResults.TestSuiteResults[CurrentSuiteNumber].Identity));
        _xml.NewParameter('name', UnitTestResults.TestSuiteResults[CurrentSuiteNumber].name);
        _xml.NewParameter('tests', UINT_TO_STRING(UnitTestResults.TestSuiteResults[CurrentSuiteNumber].NumberOfTests));
        _xml.NewParameter('failures', UINT_TO_STRING(UnitTestResults.TestSuiteResults[CurrentSuiteNumber].NumberOfFailedTests));
        _xml.NewParameter('time', LREAL_TO_STRING(UnitTestResults.TestSuiteResults[CurrentSuiteNumber].Duration));

        FOR CurrentTestCount := 1 TO UnitTestResults.TestSuiteResults[CurrentSuiteNumber].NumberOfTests BY 1 DO
            // <testcase>
            _xml.NewTag('testcase');
            _xml.NewParameter('name', UnitTestResults.TestSuiteResults[CurrentSuiteNumber].TestCaseResults[CurrentTestCount].TestName);
            _xml.NewParameter('classname', UnitTestResults.TestSuiteResults[CurrentSuiteNumber].TestCaseResults[CurrentTestCount].TestClassName);
            _xml.NewParameter('time', LREAL_TO_STRING(UnitTestResults.TestSuiteResults[CurrentSuiteNumber].TestCaseResults[CurrentTestCount].Duration));

            IF UnitTestResults.TestSuiteResults[CurrentSuiteNumber].TestCaseResults[CurrentTestCount].TestIsFailed THEN
                _xml.NewParameter('status', TEST_STATUS_FAIL);
            ELSIF UnitTestResults.TestSuiteResults[CurrentSuiteNumber].TestCaseResults[CurrentTestCount].TestIsSkipped THEN
                _xml.NewParameter('status', TEST_STATUS_SKIP);
            ELSE
                _xml.NewParameter('status', TEST_STATUS_PASS);
            END_IF

            // Determine testcase fail or success
            IF UnitTestResults.TestSuiteResults[CurrentSuiteNumber].TestCaseResults[CurrentTestCount].FailureType <> E_AssertionType.Type_UNDEFINED THEN
                (* In case of fail 
                    <failure message="Values differ" type="BYTE" />
                *)
                _xml.NewTag('failure');
                _xml.NewParameter('message', UnitTestResults.TestSuiteResults[CurrentSuiteNumber].TestCaseResults[CurrentTestCount].FailureMessage);
                _xml.NewParameter('type', F_AssertionTypeToString(UnitTestResults.TestSuiteResults[CurrentSuiteNumber].TestCaseResults[CurrentTestCount].FailureType));       
                // Close failure tag
                _xml.CloseTag();
            END_IF
            
            // Close testcase tag
            _xml.CloseTag();

        END_FOR
        // Close testsuite tag
        _xml.CloseTag();

    END_FOR
    // Close testsuites
    _xml.CloseTag();

    // Delete, open, save and close the file
    _xmlFileStream.CloseFile();

    // Clear the internal buffer
    _xml.ClearBuffer();

    // Inform user
    GVL_TcUnit.AdsMessageQueue.WriteLog(MsgCtrlMask := ADSLOG_MSGTYPE_HINT,
                                        msgFmtStr := '%s',
                                        strArg := '| ==========TEST RESULTS EXPORTED===========');

    GVL_TcUnit.AdsMessageQueue.WriteLog(MsgCtrlMask := ADSLOG_MSGTYPE_HINT,
                                        msgFmtStr :=  '| Location: %s ',
                                        strArg := GVL_Param_TcUnit.xUnitFilePath);

    GVL_TcUnit.AdsMessageQueue.WriteLog(MsgCtrlMask := ADSLOG_MSGTYPE_HINT,
                                        MsgFmtStr := '%s',
                                        StrArg := '| ======================================');
END_IF
END_METHOD

END_FUNCTION_BLOCK

// ---- POUs/FB_XmlControl.TcPOU
(*
    Organizes parsing and composing of XML data. Data can be treated as STRING or char array.
    Buffer size of file can be set via GVL_Param_TcUnit (xUnitBufferSize)
*)
FUNCTION_BLOCK FB_XmlControl
VAR
    XmlFileStream : REFERENCE TO FB_XmlFileStream;
    TagListBuffer : FB_StreamBuffer;
    Tags : T_MaxString;
    TagListSeekBuffer : FB_StreamBuffer;
    TagsSeek : STRING;
    TagBuffer : FB_StreamBuffer;
    Tag : T_MaxString;
    TagOpen: BOOL;
    TagOpenCount : INT;
    Select : UDINT;
    SearchPosition : UDINT; 
END_VAR
VAR CONSTANT
    TAG_OPEN : STRING(1) := '<';
    TAG_CLOSE : STRING(1) := '>';
    END_TAG_CLOSE : STRING(2) := '/>';
    SPACE : STRING(1) := ' ';
    EQUALS : STRING(1) := '=';
    QUOTE : STRING(1) := '"';
    BACK_SLASH : STRING(1) := '\';
    FORWARD_SLASH : STRING(1) := '/';
    OPEN_COMMENT : STRING(5) := '<!-- ';
    CLOSE_COMMENT : STRING(4) := ' -->';
    TAB : STRING(2) := '$T';
    CR_LF : STRING(4) := '$R$N';

    CR_AS_BYTE : BYTE := 13;    
    LF_AS_BYTE : BYTE := 10;
    SPACE_AS_BYTE : BYTE := 32;    

    // $OD : ASCII code for carriage return (CR)
    // $$ : to add a $R
    // $' : to add ' (apostrophe)
    // $L or $l : line feed
    // $N or $n : new line
    // $P or $p : next page
    // $R or $r : end of line
END_VAR

METHOD PRIVATE AppendIdent
VAR_INST
  indentBuffer : T_MaxString;
  i : INT;
  end : INT;
END_VAR
indentBuffer[0] := CR_AS_BYTE;
indentBuffer[1] := LF_AS_BYTE;

FOR i:=2 TO TagOpenCount
DO
  indentBuffer[i] := SPACE_AS_BYTE;
END_FOR
indentBuffer[TagOpenCount+2] := 0;

XmlFileStream.Append := indentBuffer;
END_METHOD

// Clears the contents of the entire buffer.
METHOD PUBLIC ClearBuffer
SearchPosition := 0;
TagListSeekBuffer.Length := 0;
XmlFileStream.Length := 0;
TagsSeek := '';
Tag := '';
END_METHOD

(*
    Closes a Tag:
    XML: <MyTag />'

    Method: XML.CloseTag();
*)
METHOD PUBLIC CloseTag : T_MaxString
VAR
    ClosedTag : T_MaxString;
END_VAR
TagOpenCount := TagOpenCount - 1;

IF TagOpen THEN
    XmlFileStream.Append := END_TAG_CLOSE;
    Select := TagListBuffer.FindBack(SearchString := FORWARD_SLASH);
    ClosedTag := TagListBuffer.CutOff(StartPos := Select);
    TagOpen := FALSE;
ELSE
    AppendIdent();  
    Select := TagListBuffer.FindBack(SearchString := FORWARD_SLASH);
    ClosedTag := TagListBuffer.CutOff(StartPos := Select);
    XmlFileStream.Append := TAG_OPEN;
    XmlFileStream.Append := ClosedTag;
    XmlFileStream.Append := TAG_CLOSE;
END_IF

CloseTag := ClosedTag;
END_METHOD

//FB_Init is always available implicitly and it is used primarily for initialization.
//The return value is not evaluated. For a specific influence, you can also declare the
//methods explicitly and provide additional code there with the standard initialization
//code. You can evaluate the return value.
METHOD FB_Init: BOOL
VAR_INPUT
    bInitRetains: BOOL; // TRUE: the retain variables are initialized (reset warm / reset cold)
    bInCopyCode: BOOL;  // TRUE: the instance will be copied to the copy code afterward (online change)
    xmlFileStream : REFERENCE TO FB_XmlFileStream;
END_VAR
THIS^.XmlFileStream REF= xmlFileStream;

TagListBuffer.SetBuffer(PointerToBufferAddress := ADR(Tags), SizeOfBuffer := SIZEOF(Tags));
TagListSeekBuffer.SetBuffer(PointerToBufferAddress := ADR(TagsSeek), SizeOfBuffer := SIZEOF(TagsSeek));
TagBuffer.SetBuffer(PointerToBufferAddress := ADR(Tag), SizeOfBuffer := SIZEOF(Tag));
END_METHOD

PROPERTY Length : UDINT
GET
Length := XmlFileStream.Length;
END_GET
END_PROPERTY

(*
    Adds a comment
    XML: <!-- MyComment -->

    XML.NewComment(Comment: = 'MyComment');
*)
METHOD PUBLIC NewComment
VAR_INPUT
    Comment : T_MaxString;
END_VAR
IF TagOpen THEN
    XmlFileStream.Append := TAG_CLOSE;
    TagOpen := FALSE;
END_IF;
XmlFileStream.Append := OPEN_COMMENT;
XmlFileStream.Append := Comment;
XmlFileStream.Append := CLOSE_COMMENT;
END_METHOD

(*
    Must be called after opening a new tag

    XML.NewParameter(Name: = 'ParaName', Value: = 'Value');
*)
METHOD PUBLIC NewParameter
VAR_INPUT
    Name : T_MaxString;
    Value : T_MaxString;
END_VAR
XmlFileStream.Append := SPACE;
XmlFileStream.Append := Name;
XmlFileStream.Append := EQUALS;
XmlFileStream.Append := QUOTE;
XmlFileStream.Append := Value;
XmlFileStream.Append := QUOTE;
END_METHOD

(*
    Creates a new Tag:
    XML: <MyTag>

    XML.NewTag(Name: = 'MyTag');
*)
METHOD PUBLIC NewTag
VAR_INPUT
    Name : T_MaxString;
END_VAR
IF TagOpen THEN
    XmlFileStream.Append := TAG_CLOSE;
END_IF;

TagOpenCount := TagOpenCount + 1;
AppendIdent();

XmlFileStream.Append := TAG_OPEN;
XmlFileStream.Append := Name;
TagOpen := TRUE;
TagListBuffer.Append := FORWARD_SLASH;
TagListBuffer.Append := Name;
END_METHOD

METHOD PUBLIC NewTagData
VAR_INPUT
    Data : T_MaxString;
END_VAR
XmlFileStream.Append := TAG_CLOSE;
XmlFileStream.Append := Data;
TagOpen := FALSE;
END_METHOD

(*
    Jump to the beginning of the XML data
    XML.ToStartBuffer();
*)
METHOD PUBLIC ToStartBuffer
SearchPosition := 0;
TagListSeekBuffer.Length := 0;
TagsSeek := '';
Tag := '';
END_METHOD

(*
    Add your own preffered fileheader like:
    XML: <?xml version="1.0" encoding="UTF-8"?>
    
    Start with calling this method before appending any other tags!

    XML.WriteDocumentHeader('<?xml version="1.0" encoding="UTF-8"?>');
*)
METHOD PUBLIC WriteDocumentHeader
VAR_INPUT
    Header : T_MaxString;
END_VAR
XmlFileStream.Append := Header;
END_METHOD

END_FUNCTION_BLOCK

// ---- POUs/FB_StreamBuffer.TcPOU
// This functionblock acts as a stream buffer for use with FB_XmlControl
FUNCTION_BLOCK FB_StreamBuffer 
VAR
    _PointerToStringBuffer : POINTER TO BYTE;
    _BufferSize : UDINT;
    _Length : UDINT;
END_VAR

// Appends a string to the buffer
PROPERTY Append : T_MaxString
SET
VAR
    ByteIn : POINTER TO BYTE;
    ByteBuffer : POINTER TO BYTE;
END_VAR
ByteIn := ADR(Append); 
ByteBuffer := _PointerToStringBuffer + _Length; // set start address

WHILE ByteIn^ <> 0 AND (_Length < _BufferSize ) DO
    ByteBuffer^ := ByteIn^; //Copy the 1st byte
    _Length := _Length + 1; // set new buffer length
    ByteIn := ByteIn + 1; // calculate new start address 
    ByteBuffer := ByteBuffer + 1; // calculate new start address 
END_WHILE;

ByteBuffer := _PointerToStringBuffer + _Length; // String End
ByteBuffer^ := 0; // null terminated string
END_SET
END_PROPERTY

// Read current Buffersize
PROPERTY BufferSize : UDINT
GET
BufferSize := _BufferSize;
END_GET
END_PROPERTY

// Clears the buffer and sets the length to 0
METHOD PUBLIC Clear
VAR
	Count : UDINT;
END_VAR
IF (_PointerToStringBuffer = 0) OR (_BufferSize = 0) THEN
    RETURN;
END_IF

FOR Count := 0 TO (_BufferSize - 1) DO
    _PointerToStringBuffer[Count] := 0;
END_FOR

_Length := 0;
END_METHOD

// Copies a string from the character buffer
METHOD PUBLIC Copy : T_MaxString
VAR_INPUT
    StartPos : UDINT;
    EndPos : UDINT;
END_VAR
VAR_OUTPUT
    CopyLen : UDINT;
    XmlError : E_XmlError;
END_VAR
VAR
    Loop : UDINT;
    PointerToByteToCopy : POINTER TO BYTE;
    PointerToBuffer : POINTER TO BYTE;
    CurPos : UDINT;
END_VAR
Loop := 0;
PointerToByteToCopy := ADR(Copy);
PointerToBuffer := _PointerToStringBuffer + StartPos - 1;

WHILE(Loop < SIZEOF(Copy)) AND (StartPos - 1 + Loop < _Length) AND (StartPos + Loop < EndPos) DO
    PointerToByteToCopy^ := PointerToBuffer^;
    Loop := Loop + 1;
    PointerToByteToCopy := ADR(Copy) + Loop;
    PointerToBuffer := _PointerToStringBuffer + StartPos + Loop -1;
END_WHILE;

IF Loop = SIZEOF(Copy) THEN
    XmlError := E_XmlError.ErrorStringLen;
ELSIF StartPos - 1 + Loop = _Length THEN
    XmlError := E_XmlError.ErrorMaxBufferLen;
ELSE
    XmlError := E_XmlError.OK;
END_IF;

PointerToByteToCopy^ := 0;
CopyLen :=  Loop;
END_METHOD

METHOD PUBLIC CutOff : T_MaxString
VAR_INPUT
    StartPos : UDINT;
END_VAR
VAR_OUTPUT
    CutLen : UDINT; 
    XmlError : E_XmlError;
END_VAR
VAR
    Loop : UDINT;
    PointerToByteToCut : POINTER TO BYTE;
    PointerToByteBuffer : POINTER TO BYTE;
END_VAR
Loop := 0;
PointerToByteToCut := ADR(CutOff);
PointerToByteBuffer := _PointerToStringBuffer + StartPos - 1;

WHILE PointerToByteBuffer^ <> 0 AND(Loop < SIZEOF(CutOff)) AND StartPos -1  + Loop < _Length DO
    PointerToByteToCut^ := PointerToByteBuffer^;
    Loop := Loop + 1;
    PointerToByteToCut := ADR(CutOff) + Loop;
    PointerToByteBuffer := _PointerToStringBuffer + StartPos - 1 + Loop;
END_WHILE;

IF PointerToByteBuffer^ = 0 THEN
    XmlError := E_XmlError.OK;
ELSIF Loop = SIZEOF(CutOff) THEN
    XmlError := E_XmlError.ErrorStringLen;
ELSIF StartPos - 1 + Loop = _Length THEN
    XmlError := E_XmlError.ErrorMaxBufferLen;
END_IF;

PointerToByteToCut^ := 0;
_Length := StartPos -1;

PointerToByteBuffer := _PointerToStringBuffer + StartPos - 1;
PointerToByteBuffer^ := 0;

CutLen := Loop;
END_METHOD

(* 
    Find a searchstring in the buffer and returns its position.
    It's possible to add a preffered startposition within buffer
*)
METHOD PUBLIC Find : UDINT
VAR_INPUT
    SearchString : STRING;
    StartPos : UDINT;
END_VAR
VAR
    Loop : UDINT;
    Search : UDINT;
    PointerToBuffer : POINTER TO BYTE;
    PointerToSearch : POINTER TO BYTE;
END_VAR
Loop := 0;
Search := 0;

PointerToBuffer := _PointerToStringBuffer + StartPos;
PointerToSearch := ADR(SearchString);

WHILE(PointerToSearch^ <> 0 ) AND Loop + StartPos < _Length DO
    IF PointerToBuffer^ <> PointerToSearch^ THEN
        Loop := Loop + 1;
        PointerToBuffer := _PointerToStringBuffer + StartPos + Loop;
        PointerToSearch := ADR(SearchString);
        Search := 0;
    ELSE
        Search := Search + 1;
        PointerToBuffer := _PointerToStringBuffer + StartPos + Loop + Search;
        PointerToSearch := ADR(SearchString ) + Search;
    END_IF;
END_WHILE;
Find := Loop + 1 + StartPos;
END_METHOD

METHOD PUBLIC FindBack : UDINT
VAR_INPUT
    SearchString : T_MaxString;
END_VAR
VAR
    Loop : UDINT;
    Search : UDINT;
    PointerToBuffer : POINTER TO BYTE;
    PointerToSearch : POINTER TO BYTE;
END_VAR
Loop := 0;
Search := 0;

PointerToBuffer := _PointerToStringBuffer + _Length;
PointerToSearch := ADR(SearchString);

WHILE(PointerToSearch^ <> 0) AND Loop < _Length DO
    IF PointerToBuffer^ <> PointerToSearch^ THEN
        Loop := Loop + 1;
        PointerToBuffer := _PointerToStringBuffer + _Length - Loop;
        PointerToSearch := ADR(SearchString);
        Search := 0;
    ELSE
        Search := Search + 1;
        PointerToBuffer := _PointerToStringBuffer + _Length - Loop + Search;
        PointerToSearch := ADR(SearchString ) + Search;
    END_IF;
END_WHILE;
FindBack := _Length - Loop + 1;
END_METHOD

// Gets/Sets the current length (in bytes) of the streambuffer
PROPERTY Length : UDINT
GET
Length := _Length;
END_GET
SET
_Length := Length;
END_SET
END_PROPERTY

METHOD PUBLIC SetBuffer : BOOL;
VAR_INPUT
    PointerToBufferAddress : POINTER TO BYTE; // Set buffer address (ADR ...)
    SizeOfBuffer : UDINT; // Set buffer size (SIZEOF ...)
END_VAR
IF (PointerToBufferAddress = 0) OR (SizeOfBuffer = 0) THEN
    SetBuffer := FALSE;
    RETURN;
END_IF;

_BufferSize := SizeOfBuffer;
_PointerToStringBuffer := PointerToBufferAddress;

SetBuffer := TRUE;
END_METHOD

END_FUNCTION_BLOCK

// ---- POUs/FB_TestSuite.TcPOU
(* This function block is responsible for holding the internal state of the test suite.
   Every test suite can have one or more tests, and every test can do one or more asserts.
   It's also responsible for providing all the assert-methods for asserting different data types.
   Only failed assertions are recorded.
*)
{attribute 'call_after_init'}
{attribute 'reflection'}
FUNCTION_BLOCK FB_TestSuite
VAR
    {attribute 'instance-path'}
    {attribute 'noinit'}
    InstancePath : T_MaxString;

    (* We need to have access to specific information of the current task that this test suite
       is executed in. This is for instance necessary when we need to know whether a test is
       defined already. The definition of a test that is defined already is that we call on it
       with the same name twice in the same cycle *)
    GetCurrentTaskIndex : GETCURTASKINDEX;

    NumberOfTests : UINT(0..GVL_Param_TcUnit.MaxNumberOfTestsForEachTestSuite) := 0;
    Tests : ARRAY[1..GVL_Param_TcUnit.MaxNumberOfTestsForEachTestSuite] OF FB_Test;
    (* Rising trigger of whether we have already notified the user of that the test name pointed to by the current
       position is a duplicate *)
    TestDuplicateNameTrigger : ARRAY[1..GVL_Param_TcUnit.MaxNumberOfTestsForEachTestSuite] OF R_TRIG;
    (* Last cycle count index for a specific test. Used to detect whether this test has already been defined in the
       current test suite *)
    TestCycleCountIndex : ARRAY[1..GVL_Param_TcUnit.MaxNumberOfTestsForEachTestSuite] OF UDINT;

    AssertResults : FB_AssertResultStatic;
    AssertArrayResults : FB_AssertArrayResultStatic;

    (* Prints the failed asserts to ADS so that Visual Studio can display the assert message.
       This assert formatter can be replaced with something else than ADS *)
    AdsAssertMessageFormatter : FB_AdsAssertMessageFormatter;
    AssertMessageFormatter : I_AssertMessageFormatter := AdsAssertMessageFormatter;

    (* Stores the CPU cycle count with 100ns precision. It also is an indication whether this 
       test suite has started running its tests (> 0 means it has started) *)
    StartedAt : LWORD;

    (* Duration it took to run all tests in this testsuite - including the overhead from TcUnit
       in seconds *)
    Duration : LREAL;

    // Number of ordered tests (created by TEST_ORDERED()) that this test suite contains
    NumberOfOrderedTests : UINT(0..GVL_Param_TcUnit.MaxNumberOfTestsForEachTestSuite);
END_VAR

METHOD INTERNAL AddTest : REFERENCE TO FB_Test
VAR_INPUT
    TestName : T_MaxString;
    IsTestOrdered : BOOL;
END_VAR
VAR
    IteratorCounter : UINT;
    ErrorMessage : T_MaxString;
    TestInstancePath : T_MaxString;
    FunctionCallResult : DINT;
    CycleCount : UDINT;
    TestWithThisNameAlreadyExists : BOOL := FALSE;
    LowerCasedTestName : T_MaxString;
    TrimmedTestName : T_MaxString;
    IgnoreCurrentTestCase : BOOL;
    NumberOfTestsToAnalyse : UINT(1..GVL_Param_TcUnit.MaxNumberOfTestsForEachTestSuite);
END_VAR
GVL_TcUnit.IgnoreCurrentTest := FALSE; // Reset the ignore current test flag

TrimmedTestName := F_LTrim(in := TestName);
TrimmedTestName := F_RTrim(in := TrimmedTestName);
LowerCasedTestName := F_ToLCase(in := TrimmedTestName);

// If test should be disabled, make sure to remove the "disabled_"-part of it from the test name
IF FIND(STR1 := LowerCasedTestName, STR2 := 'disabled_') = 1 THEN
    IgnoreCurrentTestCase := TRUE;
    TrimmedTestName := DELETE(STR := TrimmedTestName, LEN := LEN(STR := 'disabled_'), POS := 1);
END_IF

GetCurrentTaskIndex(); // Gets the task index of where this function block instance is being run in

(* Check if the test name already exists. Make sure there are no other tests with the same name already
   added for this test suite *)

CycleCount := TwinCAT_SystemInfoVarList._TaskInfo[GetCurrentTaskIndex.index].CycleCount;

// Limit the test analyse to the max array limit of 'Tests[]'
NumberOfTestsToAnalyse := GetNumberOfTestsToAnalyse();

// Iterate all the test names that up to this point have been added for this test suite
FOR IteratorCounter := 1 TO NumberOfTestsToAnalyse BY 1 DO
    IF Tests[IteratorCounter].GetName() = TrimmedTestName THEN
        TestWithThisNameAlreadyExists := TRUE;
        // Check if a test with this name has already been called in this PLC cycle
        IF TestCycleCountIndex[IteratorCounter] = CycleCount THEN
            GVL_TcUnit.IgnoreCurrentTest := TRUE;
            (* A test with this name already exists for this test suite and has already been called in this cycle.
               Send a message notification, but only if we have not done so already. *)
            TestDuplicateNameTrigger[IteratorCounter](CLK := TRUE);
            IF TestDuplicateNameTrigger[IteratorCounter].Q THEN // Rising edge detected. We have not reported this before
                TestInstancePath := F_RemoveInstancePathAndProjectNameFromTestInstancePath(TestInstancePath :=
                                                                                           GVL_TcUnit.CurrentTestSuiteBeingCalled^.GetInstancePath());
                ErrorMessage := 'Test with name $'%s$' already exists in test suite $'';
                ErrorMessage := CONCAT(STR1 := ErrorMessage, STR2 := TestInstancePath);
                ErrorMessage := CONCAT(STR1 := ErrorMessage, STR2 := '$'');
                GVL_TcUnit.AdsMessageQueue.WriteLog(MsgCtrlMask := ADSLOG_MSGTYPE_ERROR,
                                                    MsgFmtStr := ErrorMessage,
                                                    StrArg := TrimmedTestName);
            END_IF
        END_IF
        TestCycleCountIndex[IteratorCounter] := CycleCount;
    END_IF
END_FOR

IF NOT TestWithThisNameAlreadyExists THEN
    // Test has not been found. Add it.
    Tests[IteratorCounter].SetName(Name := TrimmedTestName);
    NumberOfTests := NumberOfTests + 1;
    TestCycleCountIndex[NumberOfTests] := CycleCount;
    IF IgnoreCurrentTestCase THEN
        Tests[IteratorCounter].SetSkipped();
    END_IF

    // Extra information to be added if test is ordered (called by TEST_ORDERED())
    IF IsTestOrdered THEN
        NumberOfOrderedTests := NumberOfOrderedTests + 1;
        Tests[IteratorCounter].SetTestOrder(OrderNumber := NumberOfOrderedTests);
    END_IF
END_IF

// Check if this test should be disabled
IF IgnoreCurrentTestCase THEN
    GVL_TcUnit.IgnoreCurrentTest := TRUE;
    RETURN;
END_IF

AddTest REF= GetTestByName(TrimmedTestName);
END_METHOD

METHOD INTERNAL AddTestNameToInstancePath : T_MaxString
VAR_INPUT
    TestInstancePath : T_MaxString;
END_VAR
VAR
    CompleteTestInstancePath : T_MaxString;
END_VAR
CompleteTestInstancePath := CONCAT(STR1 := TestInstancePath, STR2 := '@');
AddTestNameToInstancePath := CONCAT(STR1 := CompleteTestInstancePath, STR2 := GVL_TcUnit.CurrentTestNameBeingCalled);
END_METHOD

METHOD PUBLIC AreAllTestsFinished : BOOL
VAR
    Counter : UINT;
    GetCurTaskIndex : GETCURTASKINDEX;
    NumberOfTestsToAnalyse : UINT(1..GVL_Param_TcUnit.MaxNumberOfTestsForEachTestSuite);
END_VAR
AreAllTestsFinished := FALSE;

IF NumberOfTests > 0 THEN
    AreAllTestsFinished := TRUE;
    // Limit the test analyse to the max array limit of 'Tests[]'
    NumberOfTestsToAnalyse := GetNumberOfTestsToAnalyse();
    // A test is considered finished if it is finished running (i.e. set by TEST_FINISHED) or if it is skipped/disabled
    FOR Counter := 1 TO NumberOfTestsToAnalyse BY 1 DO
        AreAllTestsFinished := AreAllTestsFinished AND (Tests[Counter].IsFinished() OR Tests[Counter].IsSkipped());
    END_FOR
END_IF

(* If we have been running at least one cycle and no tests are registered, it means that this testsuite is empty
   and doesn't contain any test cases. In that case, ignore this testsuite. *)
GetCurTaskIndex();
IF NumberOfTests = 0 AND NOT TwinCAT_SystemInfoVarList._TaskInfo[GetCurTaskIndex.index].FirstCycle AND StartedAt > 0 THEN
	AreAllTestsFinished := TRUE;
END_IF
END_METHOD

// Asserts that two LREAL 2D-arrays are equal to within a positive delta. If they are not, an assertion error is created.
METHOD PUBLIC AssertArray2dEquals_LREAL
VAR_IN_OUT
    Expecteds : ARRAY[*,*] OF LREAL; // LREAL 2d array with expected values
    Actuals : ARRAY[*,*] OF LREAL; // LREAL 2d array with actual values
END_VAR
VAR_INPUT
    Delta : LREAL; // The maximum delta between the value of expected and actual for which both numbers are still considered equal, proportional to the expected value in that array cell
    Message : T_MaxString; // The identifying message for the assertion error
END_VAR
VAR
    Equals : BOOL := TRUE;
    SizeEquals : BOOL := TRUE;
    DeltaIsValid : BOOL := TRUE;
    ExpectedString : T_MaxString;
    ActualString : T_MaxString;
    AlreadyReported : BOOL;
    TestInstancePath : T_MaxString;
    DimensionIndex : USINT; // Index when looping through Dimensions
    LowerBoundExpecteds : ARRAY[1..2] OF DINT; // Lower bounds of Expecteds array in each dimension
    UpperBoundExpecteds : ARRAY[1..2] OF DINT; // Upper bounds of Expecteds array in each dimension
    LowerBoundActuals : ARRAY[1..2] OF DINT; // Lower bounds of Actuals array in each dimension
    UpperBoundActuals : ARRAY[1..2] OF DINT; // Upper bounds of Actuals array in each dimension
    SizeOfExpecteds : ARRAY[1..2] OF DINT; // Size of Expecteds array in each dimension
    SizeOfActuals : ARRAY[1..2] OF DINT; // Size of Actuals array in each dimension
    Offset : ARRAY[1..2] OF DINT; // Current Array index offsets from Lower Bound in each dimension
    ExpectedArrayIndex : ARRAY[1..2] OF DINT; // Array of current Expected array indexes when looping through arrays
    ActualArrayIndex : ARRAY[1..2] OF DINT; // Array of current Actual array indexes when looping through arrays
    Expected : LREAL; // Single expected value
    Actual : LREAL; // Single actual value
END_VAR
IF GVL_TcUnit.IgnoreCurrentTest OR GVL_TcUnit.CurrentTestIsFinished THEN
    RETURN;
END_IF

TestInstancePath := AddTestNameToInstancePath(FindTestSuiteInstancePath());

(* UPPER_BOUND and LOWER_BOUND require literals for their second parameter,
   so they can't be called in a dimension-based loop.
   Thus we copy the array dimensions into arrays which accept variable indexes *)
LowerBoundExpecteds[1] := LOWER_BOUND(Expecteds, 1);
UpperBoundExpecteds[1] := UPPER_BOUND(Expecteds, 1);
LowerBoundExpecteds[2] := LOWER_BOUND(Expecteds, 2);
UpperBoundExpecteds[2] := UPPER_BOUND(Expecteds, 2);
LowerBoundActuals[1] := LOWER_BOUND(Actuals, 1);
UpperBoundActuals[1] := UPPER_BOUND(Actuals, 1);
LowerBoundActuals[2] := LOWER_BOUND(Actuals, 2);
UpperBoundActuals[2] := UPPER_BOUND(Actuals, 2);

FOR DimensionIndex := 1 TO 2 DO
    SizeOfExpecteds[DimensionIndex] := ABS(UpperBoundExpecteds[DimensionIndex] - LowerBoundExpecteds[DimensionIndex]) + 1;
    SizeOfActuals[DimensionIndex] := ABS(UpperBoundActuals[DimensionIndex] - LowerBoundActuals[DimensionIndex]) + 1;

    IF SizeOfExpecteds[DimensionIndex] <> SizeOfActuals[DimensionIndex] THEN
        Equals := FALSE;
        SizeEquals := FALSE;
    END_IF
END_FOR

IF LrealIsNaN (Delta) THEN
    Equals := FALSE;
    DeltaIsValid := FALSE;
ELSIF SizeEquals THEN
    (* Even though we know that both arrays are equal in size, the two arrays can start at two completely different
       indexes in each dimension, which needs to be taken into account. *)
    FOR Offset[1] := 0 TO SizeOfExpecteds[1] - 1 DO // Iterate Dimension 1
        FOR Offset[2] := 0 TO SizeOfExpecteds[2] - 1 DO // Iterate Dimension 2
            // Update index variables
            FOR DimensionIndex := 1 TO 2 DO
                ExpectedArrayIndex[DimensionIndex] := LowerBoundExpecteds[DimensionIndex] + Offset[DimensionIndex];
                ActualArrayIndex[DimensionIndex] := LowerBoundActuals[DimensionIndex] + Offset[DimensionIndex];
            END_FOR

            // Get array element values
            Expected := Expecteds[ExpectedArrayIndex[1], ExpectedArrayIndex[2]];
            Actual := Actuals[ActualArrayIndex[1], ActualArrayIndex[2]]; 

            IF (LrealIsNaN (Expected)
            OR  LrealIsNaN (Actual)) THEN
                Equals := FALSE;
                EXIT;
            END_IF
            IF ABS(Expected - Actual) > Delta THEN
                Equals := FALSE;
                EXIT;
            END_IF
        END_FOR

        // Check for loop bailout
        IF NOT Equals THEN
            EXIT;
        END_IF
    END_FOR
END_IF

AssertArrayResults.ReportResult(ExpectedsSize := DINT_TO_UDINT(SizeOfExpecteds[1] * SizeOfExpecteds[2]),
                                ExpectedsTypeClass := IBaseLibrary.TypeClass.TYPE_LREAL,
                                ActualsSize := DINT_TO_UDINT(SizeOfActuals[1] * SizeOfActuals[2]),
                                ActualsTypeClass := IBaseLibrary.TypeClass.TYPE_LREAL,
                                Message := Message,
                                TestInstancePath := TestInstancePath,
                                AlreadyReported => AlreadyReported);

IF NOT AlreadyReported AND NOT Equals THEN
    SetTestFailed(AssertionType := E_AssertionType.Type_Array2D_LREAL,
                  AssertionMessage := Message);

    IF NOT SizeEquals THEN
        Message := CONCAT(STR1 := Message, STR2 := ', size of arrays not matching.');
        ExpectedString := 'SIZE = [';
        ExpectedString := CONCAT(STR1 := ExpectedString, STR2 := DINT_TO_STRING(LowerBoundExpecteds[1]));
        ExpectedString := CONCAT(STR1 := ExpectedString, STR2 := '..');
        ExpectedString := CONCAT(STR1 := ExpectedString, STR2 := DINT_TO_STRING(UpperBoundExpecteds[1]));
        ExpectedString := CONCAT(STR1 := ExpectedString, STR2 := ',');
        ExpectedString := CONCAT(STR1 := ExpectedString, STR2 := DINT_TO_STRING(LowerBoundExpecteds[2]));
        ExpectedString := CONCAT(STR1 := ExpectedString, STR2 := '..');
        ExpectedString := CONCAT(STR1 := ExpectedString, STR2 := DINT_TO_STRING(UpperBoundExpecteds[2]));
        ExpectedString := CONCAT(STR1 := ExpectedString, STR2 := '] (');
        ExpectedString := CONCAT(STR1 := ExpectedString, STR2 := DINT_TO_STRING(SizeOfExpecteds[1]));
        ExpectedString := CONCAT(STR1 := ExpectedString, STR2 := 'x');
        ExpectedString := CONCAT(STR1 := ExpectedString, STR2 := DINT_TO_STRING(SizeOfExpecteds[2]));
        ExpectedString := CONCAT(STR1 := ExpectedString, STR2 := ')');

        ActualString := 'SIZE = [';
        ActualString := CONCAT(STR1 := ActualString, STR2 := DINT_TO_STRING(LowerBoundActuals[1]));
        ActualString := CONCAT(STR1 := ActualString, STR2 := '..');
        ActualString := CONCAT(STR1 := ActualString, STR2 := DINT_TO_STRING(UpperBoundActuals[1]));
        ActualString := CONCAT(STR1 := ActualString, STR2 := ',');
        ActualString := CONCAT(STR1 := ActualString, STR2 := DINT_TO_STRING(LowerBoundActuals[2]));
        ActualString := CONCAT(STR1 := ActualString, STR2 := '..');
        ActualString := CONCAT(STR1 := ActualString, STR2 := DINT_TO_STRING(UpperBoundActuals[2]));
        ActualString := CONCAT(STR1 := ActualString, STR2 := '] (');
        ActualString := CONCAT(STR1 := ActualString, STR2 := DINT_TO_STRING(SizeOfActuals[1]));
        ActualString := CONCAT(STR1 := ActualString, STR2 := 'x');
        ActualString := CONCAT(STR1 := ActualString, STR2 := DINT_TO_STRING(SizeOfActuals[2]));
        ActualString := CONCAT(STR1 := ActualString, STR2 := ')');
    ELSIF NOT DeltaIsValid THEN
        Message := CONCAT(STR1 := Message, STR2 := ', value of delta is NaN.');
    ELSE
        ExpectedString := 'ARRAY[';
        ExpectedString := CONCAT(STR1 := ExpectedString, STR2 := DINT_TO_STRING(ExpectedArrayIndex[1]));
        ExpectedString := CONCAT(STR1 := ExpectedString, STR2 := ',');
        ExpectedString := CONCAT(STR1 := ExpectedString, STR2 := DINT_TO_STRING(ExpectedArrayIndex[2]));
        ExpectedString := CONCAT(STR1 := ExpectedString, STR2 := '] = ');
        ExpectedString := CONCAT(STR1 := ExpectedString, STR2 := LREAL_TO_STRING(Expected));

        ActualString := 'ARRAY[';
        ActualString := CONCAT(STR1 := ActualString, STR2 := DINT_TO_STRING(ActualArrayIndex[1]));
        ActualString := CONCAT(STR1 := ActualString, STR2 := ',');
        ActualString := CONCAT(STR1 := ActualString, STR2 := DINT_TO_STRING(ActualArrayIndex[2]));
        ActualString := CONCAT(STR1 := ActualString, STR2 := '] = ');
        ActualString := CONCAT(STR1 := ActualString, STR2 := LREAL_TO_STRING(Actual));
    END_IF

    AssertMessageFormatter.LogAssertFailure(Expected := ExpectedString,
                                            Actual := ActualString,
                                            Message := Message,
                                            TestInstancePath := TestInstancePath);
END_IF
END_METHOD

// Asserts that two REAL 2D-arrays are equal to within a positive delta. If they are not, an assertion error is created.
METHOD PUBLIC AssertArray2dEquals_REAL
VAR_IN_OUT
    Expecteds : ARRAY[*,*] OF REAL; // REAL 2d array with expected values
    Actuals : ARRAY[*,*] OF REAL; // REAL 2d array with actual values
END_VAR
VAR_INPUT
    Delta : REAL; // The maximum delta between the value of expected and actual for which both numbers are still considered equal, proportional to the expected value in that array cell
    Message : T_MaxString; // The identifying message for the assertion error
END_VAR
VAR
    Equals : BOOL := TRUE;
    SizeEquals : BOOL := TRUE;
    DeltaIsValid : BOOL := TRUE;
    ExpectedString : T_MaxString;
    ActualString : T_MaxString;
    AlreadyReported : BOOL;
    TestInstancePath : T_MaxString;
    DimensionIndex : USINT; // Index when looping through Dimensions
    LowerBoundExpecteds : ARRAY[1..2] OF DINT; // Lower bounds of Expecteds array in each dimension
    UpperBoundExpecteds : ARRAY[1..2] OF DINT; // Upper bounds of Expecteds array in each dimension
    LowerBoundActuals : ARRAY[1..2] OF DINT; // Lower bounds of Actuals array in each dimension
    UpperBoundActuals : ARRAY[1..2] OF DINT; // Upper bounds of Actuals array in each dimension
    SizeOfExpecteds : ARRAY[1..2] OF DINT; // Size of Expecteds array in each dimension
    SizeOfActuals : ARRAY[1..2] OF DINT; // Size of Actuals array in each dimension
    Offset : ARRAY[1..2] OF DINT; // Current Array index offsets from Lower Bound in each dimension
    ExpectedArrayIndex : ARRAY[1..2] OF DINT; // Array of current Expected array indexes when looping through arrays
    ActualArrayIndex : ARRAY[1..2] OF DINT; // Array of current Actual array indexes when looping through arrays
    Expected : REAL; // Single expected value
    Actual : REAL; // Single actual value
END_VAR
IF GVL_TcUnit.IgnoreCurrentTest OR GVL_TcUnit.CurrentTestIsFinished THEN
    RETURN;
END_IF

TestInstancePath := AddTestNameToInstancePath(FindTestSuiteInstancePath());

(* UPPER_BOUND and LOWER_BOUND require literals for their second parameter,
   so they can't be called in a dimension-based loop.
   Thus we copy the array dimensions into arrays which accept variable indexes *)
LowerBoundExpecteds[1] := LOWER_BOUND(Expecteds, 1);
UpperBoundExpecteds[1] := UPPER_BOUND(Expecteds, 1);
LowerBoundExpecteds[2] := LOWER_BOUND(Expecteds, 2);
UpperBoundExpecteds[2] := UPPER_BOUND(Expecteds, 2);
LowerBoundActuals[1] := LOWER_BOUND(Actuals, 1);
UpperBoundActuals[1] := UPPER_BOUND(Actuals, 1);
LowerBoundActuals[2] := LOWER_BOUND(Actuals, 2);
UpperBoundActuals[2] := UPPER_BOUND(Actuals, 2);

FOR DimensionIndex := 1 TO 2 DO
    SizeOfExpecteds[DimensionIndex] := ABS(UpperBoundExpecteds[DimensionIndex] - LowerBoundExpecteds[DimensionIndex]) + 1;
    SizeOfActuals[DimensionIndex] := ABS(UpperBoundActuals[DimensionIndex] - LowerBoundActuals[DimensionIndex]) + 1;

    IF SizeOfExpecteds[DimensionIndex] <> SizeOfActuals[DimensionIndex] THEN
        Equals := FALSE;
        SizeEquals := FALSE;
    END_IF
END_FOR

IF RealIsNaN (Delta) THEN
    Equals := FALSE;
    DeltaIsValid := FALSE;
ELSIF SizeEquals THEN
    (* Even though we know that both arrays are equal in size, the two arrays can start at two completely different
       indexes in each dimension, which needs to be taken into account. *)
    FOR Offset[1] := 0 TO SizeOfExpecteds[1] - 1 DO // Iterate Dimension 1
        FOR Offset[2] := 0 TO SizeOfExpecteds[2] - 1 DO // Iterate Dimension 2
            // Update index variables
            FOR DimensionIndex := 1 TO 2 DO
                ExpectedArrayIndex[DimensionIndex] := LowerBoundExpecteds[DimensionIndex] + Offset[DimensionIndex];
                ActualArrayIndex[DimensionIndex] := LowerBoundActuals[DimensionIndex] + Offset[DimensionIndex];
            END_FOR

            // Get array element values
            Expected := Expecteds[ExpectedArrayIndex[1], ExpectedArrayIndex[2]];
            Actual := Actuals[ActualArrayIndex[1], ActualArrayIndex[2]]; 

            IF (RealIsNaN (Expected)
            OR  RealIsNaN (Actual)) THEN
                Equals := FALSE;
                EXIT;
            END_IF
            IF ABS(Expected - Actual) > Delta THEN
                Equals := FALSE;
                EXIT;
            END_IF
        END_FOR

        // Check for loop bailout
        IF NOT Equals THEN
            EXIT;
        END_IF
    END_FOR
END_IF

AssertArrayResults.ReportResult(ExpectedsSize := DINT_TO_UDINT(SizeOfExpecteds[1] * SizeOfExpecteds[2]),
                                ExpectedsTypeClass := IBaseLibrary.TypeClass.TYPE_REAL,
                                ActualsSize := DINT_TO_UDINT(SizeOfActuals[1] * SizeOfActuals[2]),
                                ActualsTypeClass := IBaseLibrary.TypeClass.TYPE_REAL,
                                Message := Message,
                                TestInstancePath := TestInstancePath,
                                AlreadyReported => AlreadyReported);

IF NOT AlreadyReported AND NOT Equals THEN
    SetTestFailed(AssertionType := E_AssertionType.Type_Array2D_REAL,
                  AssertionMessage := Message);

    IF NOT SizeEquals THEN
        Message := CONCAT(STR1 := Message, STR2 := ', size of arrays not matching.');
        ExpectedString := 'SIZE = [';
        ExpectedString := CONCAT(STR1 := ExpectedString, STR2 := DINT_TO_STRING(LowerBoundExpecteds[1]));
        ExpectedString := CONCAT(STR1 := ExpectedString, STR2 := '..');
        ExpectedString := CONCAT(STR1 := ExpectedString, STR2 := DINT_TO_STRING(UpperBoundExpecteds[1]));
        ExpectedString := CONCAT(STR1 := ExpectedString, STR2 := ',');
        ExpectedString := CONCAT(STR1 := ExpectedString, STR2 := DINT_TO_STRING(LowerBoundExpecteds[2]));
        ExpectedString := CONCAT(STR1 := ExpectedString, STR2 := '..');
        ExpectedString := CONCAT(STR1 := ExpectedString, STR2 := DINT_TO_STRING(UpperBoundExpecteds[2]));
        ExpectedString := CONCAT(STR1 := ExpectedString, STR2 := '] (');
        ExpectedString := CONCAT(STR1 := ExpectedString, STR2 := DINT_TO_STRING(SizeOfExpecteds[1]));
        ExpectedString := CONCAT(STR1 := ExpectedString, STR2 := 'x');
        ExpectedString := CONCAT(STR1 := ExpectedString, STR2 := DINT_TO_STRING(SizeOfExpecteds[2]));
        ExpectedString := CONCAT(STR1 := ExpectedString, STR2 := ')');

        ActualString := 'SIZE = [';
        ActualString := CONCAT(STR1 := ActualString, STR2 := DINT_TO_STRING(LowerBoundActuals[1]));
        ActualString := CONCAT(STR1 := ActualString, STR2 := '..');
        ActualString := CONCAT(STR1 := ActualString, STR2 := DINT_TO_STRING(UpperBoundActuals[1]));
        ActualString := CONCAT(STR1 := ActualString, STR2 := ',');
        ActualString := CONCAT(STR1 := ActualString, STR2 := DINT_TO_STRING(LowerBoundActuals[2]));
        ActualString := CONCAT(STR1 := ActualString, STR2 := '..');
        ActualString := CONCAT(STR1 := ActualString, STR2 := DINT_TO_STRING(UpperBoundActuals[2]));
        ActualString := CONCAT(STR1 := ActualString, STR2 := '] (');
        ActualString := CONCAT(STR1 := ActualString, STR2 := DINT_TO_STRING(SizeOfActuals[1]));
        ActualString := CONCAT(STR1 := ActualString, STR2 := 'x');
        ActualString := CONCAT(STR1 := ActualString, STR2 := DINT_TO_STRING(SizeOfActuals[2]));
        ActualString := CONCAT(STR1 := ActualString, STR2 := ')');
    ELSIF NOT DeltaIsValid THEN
        Message := CONCAT(STR1 := Message, STR2 := ', value of delta is NaN.');
    ELSE
        ExpectedString := 'ARRAY[';
        ExpectedString := CONCAT(STR1 := ExpectedString, STR2 := DINT_TO_STRING(ExpectedArrayIndex[1]));
        ExpectedString := CONCAT(STR1 := ExpectedString, STR2 := ',');
        ExpectedString := CONCAT(STR1 := ExpectedString, STR2 := DINT_TO_STRING(ExpectedArrayIndex[2]));
        ExpectedString := CONCAT(STR1 := ExpectedString, STR2 := '] = ');
        ExpectedString := CONCAT(STR1 := ExpectedString, STR2 := REAL_TO_STRING(Expected));

        ActualString := 'ARRAY[';
        ActualString := CONCAT(STR1 := ActualString, STR2 := DINT_TO_STRING(ActualArrayIndex[1]));
        ActualString := CONCAT(STR1 := ActualString, STR2 := ',');
        ActualString := CONCAT(STR1 := ActualString, STR2 := DINT_TO_STRING(ActualArrayIndex[2]));
        ActualString := CONCAT(STR1 := ActualString, STR2 := '] = ');
        ActualString := CONCAT(STR1 := ActualString, STR2 := REAL_TO_STRING(Actual));
    END_IF

    AssertMessageFormatter.LogAssertFailure(Expected := ExpectedString,
                                            Actual := ActualString,
                                            Message := Message,
                                            TestInstancePath := TestInstancePath);
END_IF
END_METHOD

// Asserts that two LREAL 3D-arrays are equal to within a positive delta. If they are not, an assertion error is created.
METHOD PUBLIC AssertArray3dEquals_LREAL
VAR_IN_OUT
    Expecteds : ARRAY[*,*,*] OF LREAL; // LREAL 3d array with expected values
    Actuals : ARRAY[*,*,*] OF LREAL; // LREAL 3d array with actual values
END_VAR
VAR_INPUT
    Delta : LREAL; // The maximum delta between the value of expected and actual for which both numbers are still considered equal, proportional to the expected value in that array cell
    Message : T_MaxString; // The identifying message for the assertion error
END_VAR
VAR
    Equals : BOOL := TRUE;
    SizeEquals : BOOL := TRUE;
    DeltaIsValid : BOOL := TRUE;
    ExpectedString : T_MaxString;
    ActualString : T_MaxString;
    AlreadyReported : BOOL;
    TestInstancePath : T_MaxString;
    DimensionIndex : USINT;  // Index when looping through Dimensions
    LowerBoundExpecteds : ARRAY[1..3] OF DINT; // Lower bounds of Expecteds array in each dimension
    UpperBoundExpecteds : ARRAY[1..3] OF DINT; // Upper bounds of Expecteds array in each dimension
    LowerBoundActuals : ARRAY[1..3] OF DINT; // Lower bounds of Actuals array in each dimension
    UpperBoundActuals : ARRAY[1..3] OF DINT; // Upper bounds of Actuals array in each dimension
    SizeOfExpecteds : ARRAY[1..3] OF DINT; // Size of Expecteds array in each dimension
    SizeOfActuals : ARRAY[1..3] OF DINT; // Size of Actuals array in each dimension
    Offset : ARRAY[1..3] OF DINT; // Current Array index offsets from Lower Bound in each dimension
    ExpectedArrayIndex : ARRAY[1..3] OF DINT; // Array of current Expected array indexes when looping through arrays
    ActualArrayIndex : ARRAY[1..3] OF DINT; // Array of current Actual array indexes when looping through arrays
    Expected : LREAL; // Single expected value
    Actual : LREAL; // Single actual value
END_VAR
IF GVL_TcUnit.IgnoreCurrentTest OR GVL_TcUnit.CurrentTestIsFinished THEN
    RETURN;
END_IF

TestInstancePath := AddTestNameToInstancePath(FindTestSuiteInstancePath());

(* UPPER_BOUND and LOWER_BOUND require literals for their second parameter,
   so they can't be called in a dimension-based loop.
   Thus we copy the array dimensions into arrays which accept variable indexes *)
LowerBoundExpecteds[1] := LOWER_BOUND(Expecteds, 1);
UpperBoundExpecteds[1] := UPPER_BOUND(Expecteds, 1);
LowerBoundExpecteds[2] := LOWER_BOUND(Expecteds, 2);
UpperBoundExpecteds[2] := UPPER_BOUND(Expecteds, 2);
LowerBoundExpecteds[3] := LOWER_BOUND(Expecteds, 3);
UpperBoundExpecteds[3] := UPPER_BOUND(Expecteds, 3);
LowerBoundActuals[1] := LOWER_BOUND(Actuals, 1);
UpperBoundActuals[1] := UPPER_BOUND(Actuals, 1);
LowerBoundActuals[2] := LOWER_BOUND(Actuals, 2);
UpperBoundActuals[2] := UPPER_BOUND(Actuals, 2);
LowerBoundActuals[3] := LOWER_BOUND(Actuals, 3);
UpperBoundActuals[3] := UPPER_BOUND(Actuals, 3);

FOR DimensionIndex := 1 TO 3 DO
    SizeOfExpecteds[DimensionIndex] := ABS(UpperBoundExpecteds[DimensionIndex] - LowerBoundExpecteds[DimensionIndex]) + 1;
    SizeOfActuals[DimensionIndex] := ABS(UpperBoundActuals[DimensionIndex] - LowerBoundActuals[DimensionIndex]) + 1;

    IF SizeOfExpecteds[DimensionIndex] <> SizeOfActuals[DimensionIndex] THEN
        Equals := FALSE;
        SizeEquals := FALSE;
    END_IF
END_FOR

